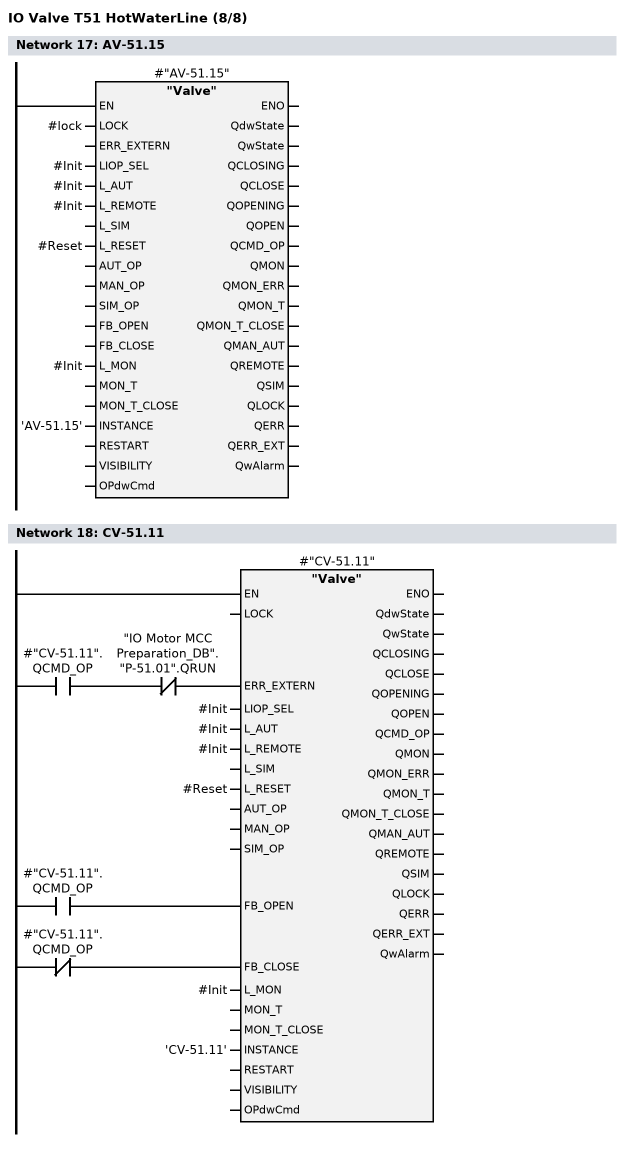
   RUNG wire#powerrail
      #"AV-51.15"(LOCK := #lock, ERR_EXTERN :=, LIOP_SEL := #Init, L_AUT := #Init, L_REMOTE := #Init, L_SIM :=, L_RESET := #Reset, AUT_OP :=, MAN_OP :=, SIM_OP :=, FB_OPEN :=, FB_CLOSE :=, L_MON := #Init, MON_T :=, MON_T_CLOSE :=, INSTANCE := 'AV-51.15', RESTART :=, VISIBILITY :=, OPdwCmd :=, QdwState =>, QwState =>, QCLOSING =>, QCLOSE =>, QOPENING =>, QOPEN =>, QCMD_OP =>, QMON =>, QMON_ERR =>, QMON_T =>, QMON_T_CLOSE =>, QMAN_AUT =>, QREMOTE =>, QSIM =>, QLOCK =>, QERR =>, QERR_EXT =>, QwAlarm =>)
   END_RUNG
   // the same network as SCL:
   #"AV-51.15"(LOCK := #lock,   // "Valve"
               LIOP_SEL := #Init,
               L_AUT := #Init,
               L_REMOTE := #Init,
               L_RESET := #Reset,
               L_MON := #Init,
               INSTANCE := 'AV-51.15');
END_REGION

REGION Network 18: CV-51.11
   RUNG wire#powerrail
      #"CV-51.11"(ERR_EXTERN := wire#w1, FB_OPEN := wire#w2, FB_CLOSE := wire#w3, LOCK :=, LIOP_SEL := #Init, L_AUT := #Init, L_REMOTE := #Init, L_SIM :=, L_RESET := #Reset, AUT_OP :=, MAN_OP :=, SIM_OP :=, L_MON := #Init, MON_T :=, MON_T_CLOSE :=, INSTANCE := 'CV-51.11', RESTART :=, VISIBILITY :=, OPdwCmd :=, QdwState =>, QwState =>, QCLOSING =>, QCLOSE =>, QOPENING =>, QOPEN =>, QCMD_OP =>, QMON =>, QMON_ERR =>, QMON_T =>, QMON_T_CLOSE =>, QMAN_AUT =>, QREMOTE =>, QSIM =>, QLOCK =>, QERR =>, QERR_EXT =>, QwAlarm =>)
   END_RUNG
   RUNG wire#powerrail
      Contact( #"CV-51.11".QCMD_OP )
      I_Contact( "IO Motor MCC Preparation_DB"."P-51.01".QRUN )
   END_RUNG wire#w1
   RUNG wire#powerrail
      Contact( #"CV-51.11".QCMD_OP )
   END_RUNG wire#w2
   RUNG wire#powerrail
      I_Contact( #"CV-51.11".QCMD_OP )
   END_RUNG wire#w3
   // the same network as SCL:
   #"CV-51.11"(ERR_EXTERN := #"CV-51.11".QCMD_OP AND NOT "IO Motor MCC Preparation_DB"."P-51.01".QRUN,   // "Valve"
               LIOP_SEL := #Init,
               L_AUT := #Init,
               L_REMOTE := #Init,
               L_RESET := #Reset,
               FB_OPEN := #"CV-51.11".QCMD_OP,
               FB_CLOSE := NOT #"CV-51.11".QCMD_OP,
               L_MON := #Init,
               INSTANCE := 'CV-51.11');
END_REGION
END_FUNCTION_BLOCK

FUNCTION "IO Homoge" : Void   // FC1, LAD
{ S7_Optimized_Access := 'TRUE' }
VERSION : 0.1
// stored: AutoNumber true, IsIECCheckEnabled false, SetENOAutomatically false, UDAEnableTagReadback false
BEGIN

REGION Network 1: Analog
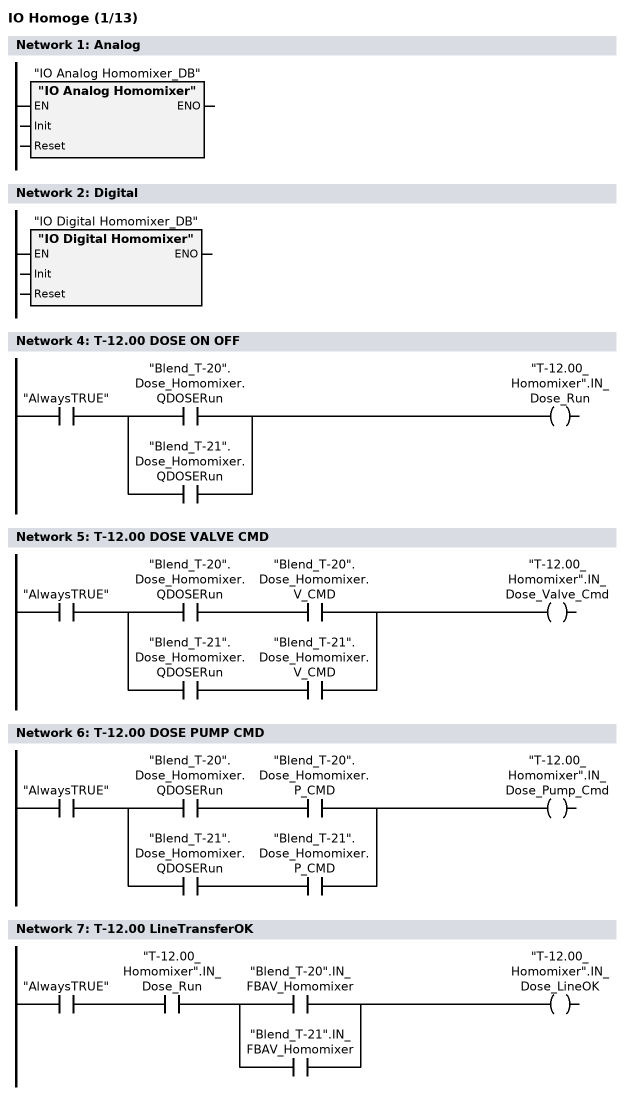
   RUNG wire#powerrail
      "IO Analog Homomixer_DB"(Init :=, Reset :=)
   END_RUNG
   // the same network as SCL:
   "IO Analog Homomixer_DB"();   // "IO Analog Homomixer"
END_REGION

REGION Network 2: Digital
   RUNG wire#powerrail
      "IO Digital Homomixer_DB"(Init :=, Reset :=)
   END_RUNG
   // the same network as SCL:
   "IO Digital Homomixer_DB"();   // "IO Digital Homomixer"
END_REGION

REGION Network 4: T-12.00 DOSE ON OFF
   RUNG wire#powerrail
      Contact( "AlwaysTRUE" )
      wire#w1
      Contact( "Blend_T-20".Dose_Homomixer.QDOSERun )
      wire#w2
      Coil( "T-12.00_Homomixer".IN_Dose_Run )
   END_RUNG
   RUNG wire#w1
      Contact( "Blend_T-21".Dose_Homomixer.QDOSERun )
   END_RUNG wire#w2
   // the same network as SCL:
   "T-12.00_Homomixer".IN_Dose_Run := "AlwaysTRUE" AND ("Blend_T-20".Dose_Homomixer.QDOSERun OR "Blend_T-21".Dose_Homomixer.QDOSERun);
END_REGION

REGION Network 5: T-12.00 DOSE VALVE CMD
   RUNG wire#powerrail
      Contact( "AlwaysTRUE" )
      wire#w1
      Contact( "Blend_T-20".Dose_Homomixer.QDOSERun )
      Contact( "Blend_T-20".Dose_Homomixer.V_CMD )
      wire#w2
      Coil( "T-12.00_Homomixer".IN_Dose_Valve_Cmd )
   END_RUNG
   RUNG wire#w1
      Contact( "Blend_T-21".Dose_Homomixer.QDOSERun )
      Contact( "Blend_T-21".Dose_Homomixer.V_CMD )
   END_RUNG wire#w2
   // the same network as SCL:
   "T-12.00_Homomixer".IN_Dose_Valve_Cmd := "AlwaysTRUE" AND (("Blend_T-20".Dose_Homomixer.QDOSERun AND "Blend_T-20".Dose_Homomixer.V_CMD) OR ("Blend_T-21".Dose_Homomixer.QDOSERun AND "Blend_T-21".Dose_Homomixer.V_CMD));
END_REGION

REGION Network 6: T-12.00 DOSE PUMP CMD
   RUNG wire#powerrail
      Contact( "AlwaysTRUE" )
      wire#w1
      Contact( "Blend_T-20".Dose_Homomixer.QDOSERun )
      Contact( "Blend_T-20".Dose_Homomixer.P_CMD )
      wire#w2
      Coil( "T-12.00_Homomixer".IN_Dose_Pump_Cmd )
   END_RUNG
   RUNG wire#w1
      Contact( "Blend_T-21".Dose_Homomixer.QDOSERun )
      Contact( "Blend_T-21".Dose_Homomixer.P_CMD )
   END_RUNG wire#w2
   // the same network as SCL:
   "T-12.00_Homomixer".IN_Dose_Pump_Cmd := "AlwaysTRUE" AND (("Blend_T-20".Dose_Homomixer.QDOSERun AND "Blend_T-20".Dose_Homomixer.P_CMD) OR ("Blend_T-21".Dose_Homomixer.QDOSERun AND "Blend_T-21".Dose_Homomixer.P_CMD));
END_REGION

REGION Network 7: T-12.00 LineTransferOK
   RUNG wire#powerrail
      Contact( "AlwaysTRUE" )
      Contact( "T-12.00_Homomixer".IN_Dose_Run )
      wire#w1
      Contact( "Blend_T-20".IN_FBAV_Homomixer )
      wire#w2
      Coil( "T-12.00_Homomixer".IN_Dose_LineOK )
   END_RUNG
   RUNG wire#w1
      Contact( "Blend_T-21".IN_FBAV_Homomixer )
   END_RUNG wire#w2
   // the same network as SCL:
   "T-12.00_Homomixer".IN_Dose_LineOK := "AlwaysTRUE" AND "T-12.00_Homomixer".IN_Dose_Run AND ("Blend_T-20".IN_FBAV_Homomixer OR "Blend_T-21".IN_FBAV_Homomixer);
END_REGION

REGION Network 8: T-12.00 Homomixer
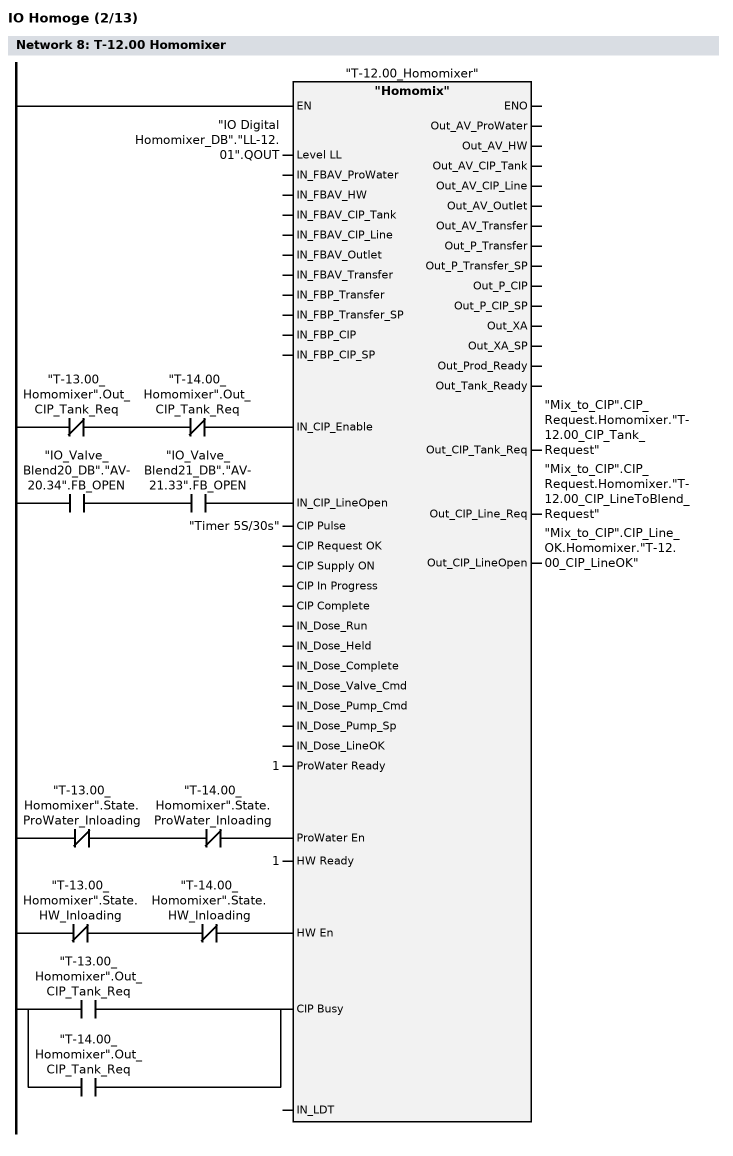
   RUNG wire#powerrail
      "T-12.00_Homomixer"(IN_CIP_Enable := wire#w1, IN_CIP_LineOpen := wire#w2, "ProWater En" := wire#w3, "HW En" := wire#w4, "CIP Busy" := wire#w5, "Level LL" := "IO Digital Homomixer_DB"."LL-12.01".QOUT, IN_FBAV_ProWater :=, IN_FBAV_HW :=, IN_FBAV_CIP_Tank :=, IN_FBAV_CIP_Line :=, IN_FBAV_Outlet :=, IN_FBAV_Transfer :=, IN_FBP_Transfer :=, IN_FBP_Transfer_SP :=, IN_FBP_CIP :=, IN_FBP_CIP_SP :=, "CIP Pulse" := "Timer 5S/30s", "CIP Request OK" :=, "CIP Supply ON" :=, "CIP In Progress" :=, "CIP Complete" :=, IN_Dose_Run :=, IN_Dose_Held :=, IN_Dose_Complete :=, IN_Dose_Valve_Cmd :=, IN_Dose_Pump_Cmd :=, IN_Dose_Pump_Sp :=, IN_Dose_LineOK :=, "ProWater Ready" := 1, "HW Ready" := 1, IN_LDT :=, Out_AV_ProWater =>, Out_AV_HW =>, Out_AV_CIP_Tank =>, Out_AV_CIP_Line =>, Out_AV_Outlet =>, Out_AV_Transfer =>, Out_P_Transfer =>, Out_P_Transfer_SP =>, Out_P_CIP =>, Out_P_CIP_SP =>, Out_XA =>, Out_XA_SP =>, Out_Prod_Ready =>, Out_Tank_Ready =>, Out_CIP_Tank_Req => "Mix_to_CIP".CIP_Request.Homomixer."T-12.00_CIP_Tank_Request", Out_CIP_Line_Req => "Mix_to_CIP".CIP_Request.Homomixer."T-12.00_CIP_LineToBlend_Request", Out_CIP_LineOpen => "Mix_to_CIP".CIP_Line_OK.Homomixer."T-12.00_CIP_LineOK")
   END_RUNG
   RUNG wire#powerrail
      I_Contact( "T-13.00_Homomixer".Out_CIP_Tank_Req )
      I_Contact( "T-14.00_Homomixer".Out_CIP_Tank_Req )
   END_RUNG wire#w1
   RUNG wire#powerrail
      Contact( "IO_Valve_Blend20_DB"."AV-20.34".FB_OPEN )
      Contact( "IO_Valve_Blend21_DB"."AV-21.33".FB_OPEN )
   END_RUNG wire#w2
   RUNG wire#powerrail
      I_Contact( "T-13.00_Homomixer".State.ProWater_Inloading )
      I_Contact( "T-14.00_Homomixer".State.ProWater_Inloading )
   END_RUNG wire#w3
   RUNG wire#powerrail
      I_Contact( "T-13.00_Homomixer".State.HW_Inloading )
      I_Contact( "T-14.00_Homomixer".State.HW_Inloading )
   END_RUNG wire#w4
   RUNG wire#powerrail
      Contact( "T-13.00_Homomixer".Out_CIP_Tank_Req )
   END_RUNG wire#w5
   RUNG wire#powerrail
      Contact( "T-14.00_Homomixer".Out_CIP_Tank_Req )
   END_RUNG wire#w5
   // the same network as SCL:
   "T-12.00_Homomixer"("Level LL" := "IO Digital Homomixer_DB"."LL-12.01".QOUT,   // "Homomix"
                       IN_CIP_Enable := NOT "T-13.00_Homomixer".Out_CIP_Tank_Req AND NOT "T-14.00_Homomixer".Out_CIP_Tank_Req,
                       IN_CIP_LineOpen := "IO_Valve_Blend20_DB"."AV-20.34".FB_OPEN AND "IO_Valve_Blend21_DB"."AV-21.33".FB_OPEN,
                       "CIP Pulse" := "Timer 5S/30s",
                       "ProWater Ready" := 1,
                       "ProWater En" := NOT "T-13.00_Homomixer".State.ProWater_Inloading AND NOT "T-14.00_Homomixer".State.ProWater_Inloading,
                       "HW Ready" := 1,
                       "HW En" := NOT "T-13.00_Homomixer".State.HW_Inloading AND NOT "T-14.00_Homomixer".State.HW_Inloading,
                       "CIP Busy" := "T-13.00_Homomixer".Out_CIP_Tank_Req OR "T-14.00_Homomixer".Out_CIP_Tank_Req,
                       Out_CIP_Tank_Req => "Mix_to_CIP".CIP_Request.Homomixer."T-12.00_CIP_Tank_Request",
                       Out_CIP_Line_Req => "Mix_to_CIP".CIP_Request.Homomixer."T-12.00_CIP_LineToBlend_Request",
                       Out_CIP_LineOpen => "Mix_to_CIP".CIP_Line_OK.Homomixer."T-12.00_CIP_LineOK");
END_REGION

REGION Network 9: T-12.00 Valve Cmd
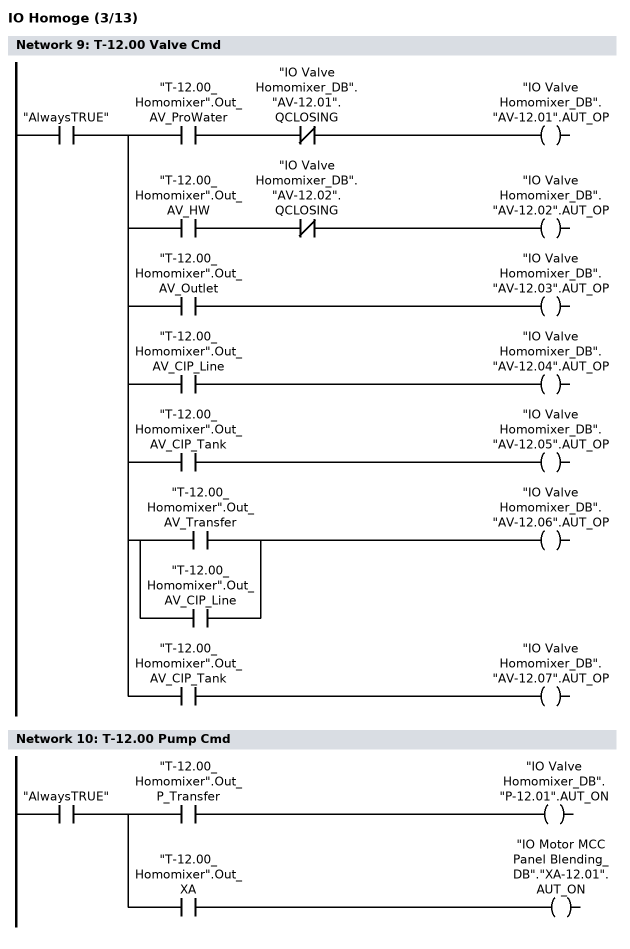
   RUNG wire#powerrail
      Contact( "AlwaysTRUE" )
      wire#w1
      Contact( "T-12.00_Homomixer".Out_AV_ProWater )
      I_Contact( "IO Valve Homomixer_DB"."AV-12.01".QCLOSING )
      Coil( "IO Valve Homomixer_DB"."AV-12.01".AUT_OP )
   END_RUNG
   RUNG wire#w1
      Contact( "T-12.00_Homomixer".Out_AV_HW )
      I_Contact( "IO Valve Homomixer_DB"."AV-12.02".QCLOSING )
      Coil( "IO Valve Homomixer_DB"."AV-12.02".AUT_OP )
   END_RUNG
   RUNG wire#w1
      Contact( "T-12.00_Homomixer".Out_AV_Outlet )
      Coil( "IO Valve Homomixer_DB"."AV-12.03".AUT_OP )
   END_RUNG
   RUNG wire#w1
      Contact( "T-12.00_Homomixer".Out_AV_CIP_Line )
      Coil( "IO Valve Homomixer_DB"."AV-12.04".AUT_OP )
   END_RUNG
   RUNG wire#w1
      Contact( "T-12.00_Homomixer".Out_AV_CIP_Tank )
      Coil( "IO Valve Homomixer_DB"."AV-12.05".AUT_OP )
   END_RUNG
   RUNG wire#w1
      Contact( "T-12.00_Homomixer".Out_AV_Transfer )
      wire#w2
      Coil( "IO Valve Homomixer_DB"."AV-12.06".AUT_OP )
   END_RUNG
   RUNG wire#w1
      Contact( "T-12.00_Homomixer".Out_AV_CIP_Line )
   END_RUNG wire#w2
   RUNG wire#w1
      Contact( "T-12.00_Homomixer".Out_AV_CIP_Tank )
      Coil( "IO Valve Homomixer_DB"."AV-12.07".AUT_OP )
   END_RUNG
   // the same network as SCL:
   "IO Valve Homomixer_DB"."AV-12.01".AUT_OP := "AlwaysTRUE" AND "T-12.00_Homomixer".Out_AV_ProWater AND NOT "IO Valve Homomixer_DB"."AV-12.01".QCLOSING;
   "IO Valve Homomixer_DB"."AV-12.02".AUT_OP := "AlwaysTRUE" AND "T-12.00_Homomixer".Out_AV_HW AND NOT "IO Valve Homomixer_DB"."AV-12.02".QCLOSING;
   "IO Valve Homomixer_DB"."AV-12.03".AUT_OP := "AlwaysTRUE" AND "T-12.00_Homomixer".Out_AV_Outlet;
   "IO Valve Homomixer_DB"."AV-12.04".AUT_OP := "AlwaysTRUE" AND "T-12.00_Homomixer".Out_AV_CIP_Line;
   "IO Valve Homomixer_DB"."AV-12.05".AUT_OP := "AlwaysTRUE" AND "T-12.00_Homomixer".Out_AV_CIP_Tank;
   "IO Valve Homomixer_DB"."AV-12.06".AUT_OP := "AlwaysTRUE" AND ("T-12.00_Homomixer".Out_AV_Transfer OR "T-12.00_Homomixer".Out_AV_CIP_Line);
   "IO Valve Homomixer_DB"."AV-12.07".AUT_OP := "AlwaysTRUE" AND "T-12.00_Homomixer".Out_AV_CIP_Tank;
END_REGION

REGION Network 10: T-12.00 Pump Cmd
   RUNG wire#powerrail
      Contact( "AlwaysTRUE" )
      wire#w1
      Contact( "T-12.00_Homomixer".Out_P_Transfer )
      Coil( "IO Valve Homomixer_DB"."P-12.01".AUT_ON )
   END_RUNG
   RUNG wire#w1
      Contact( "T-12.00_Homomixer".Out_XA )
      Coil( "IO Motor MCC Panel Blending_DB"."XA-12.01".AUT_ON )
   END_RUNG
   // the same network as SCL:
   "IO Valve Homomixer_DB"."P-12.01".AUT_ON := "AlwaysTRUE" AND "T-12.00_Homomixer".Out_P_Transfer;
   "IO Motor MCC Panel Blending_DB"."XA-12.01".AUT_ON := "AlwaysTRUE" AND "T-12.00_Homomixer".Out_XA;
END_REGION

REGION Network 11: T-12.00 Feedback Instrument
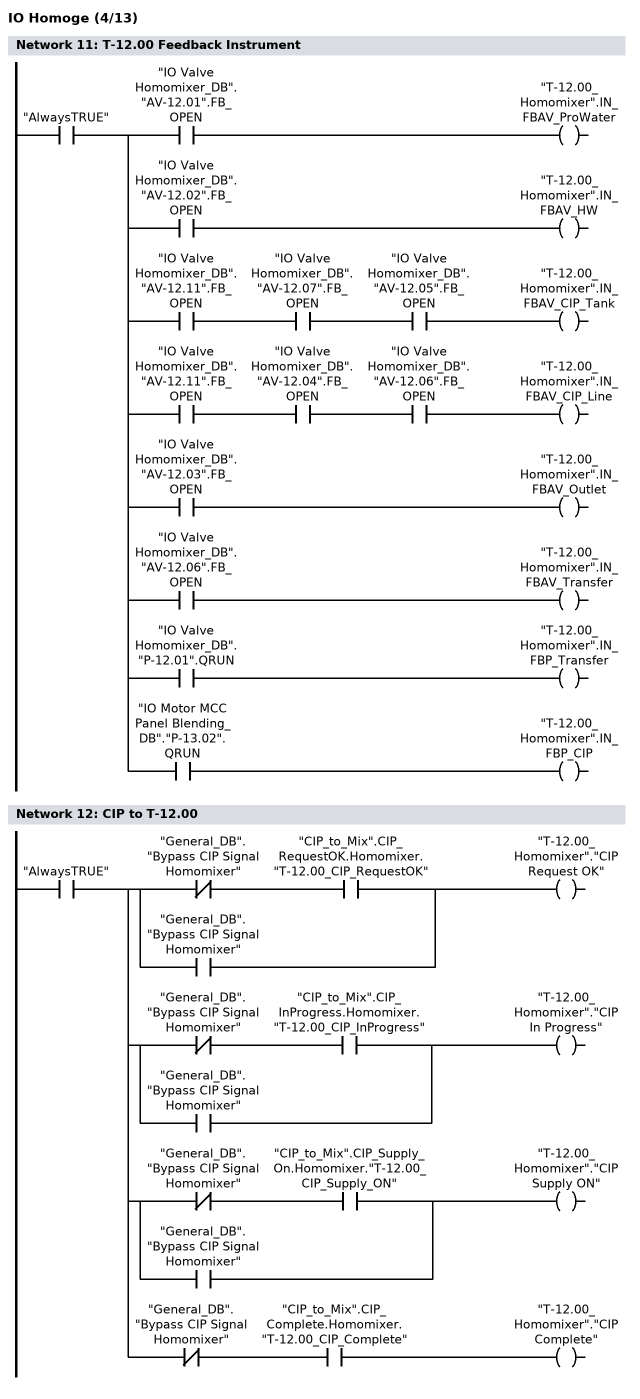
   RUNG wire#powerrail
      Contact( "AlwaysTRUE" )
      wire#w1
      Contact( "IO Valve Homomixer_DB"."AV-12.01".FB_OPEN )
      Coil( "T-12.00_Homomixer".IN_FBAV_ProWater )
   END_RUNG
   RUNG wire#w1
      Contact( "IO Valve Homomixer_DB"."AV-12.02".FB_OPEN )
      Coil( "T-12.00_Homomixer".IN_FBAV_HW )
   END_RUNG
   RUNG wire#w1
      Contact( "IO Valve Homomixer_DB"."AV-12.11".FB_OPEN )
      Contact( "IO Valve Homomixer_DB"."AV-12.07".FB_OPEN )
      Contact( "IO Valve Homomixer_DB"."AV-12.05".FB_OPEN )
      Coil( "T-12.00_Homomixer".IN_FBAV_CIP_Tank )
   END_RUNG
   RUNG wire#w1
      Contact( "IO Valve Homomixer_DB"."AV-12.11".FB_OPEN )
      Contact( "IO Valve Homomixer_DB"."AV-12.04".FB_OPEN )
      Contact( "IO Valve Homomixer_DB"."AV-12.06".FB_OPEN )
      Coil( "T-12.00_Homomixer".IN_FBAV_CIP_Line )
   END_RUNG
   RUNG wire#w1
      Contact( "IO Valve Homomixer_DB"."AV-12.03".FB_OPEN )
      Coil( "T-12.00_Homomixer".IN_FBAV_Outlet )
   END_RUNG
   RUNG wire#w1
      Contact( "IO Valve Homomixer_DB"."AV-12.06".FB_OPEN )
      Coil( "T-12.00_Homomixer".IN_FBAV_Transfer )
   END_RUNG
   RUNG wire#w1
      Contact( "IO Valve Homomixer_DB"."P-12.01".QRUN )
      Coil( "T-12.00_Homomixer".IN_FBP_Transfer )
   END_RUNG
   RUNG wire#w1
      Contact( "IO Motor MCC Panel Blending_DB"."P-13.02".QRUN )
      Coil( "T-12.00_Homomixer".IN_FBP_CIP )
   END_RUNG
   // the same network as SCL:
   "T-12.00_Homomixer".IN_FBAV_ProWater := "AlwaysTRUE" AND "IO Valve Homomixer_DB"."AV-12.01".FB_OPEN;
   "T-12.00_Homomixer".IN_FBAV_HW := "AlwaysTRUE" AND "IO Valve Homomixer_DB"."AV-12.02".FB_OPEN;
   "T-12.00_Homomixer".IN_FBAV_CIP_Tank := "AlwaysTRUE" AND "IO Valve Homomixer_DB"."AV-12.11".FB_OPEN AND "IO Valve Homomixer_DB"."AV-12.07".FB_OPEN AND "IO Valve Homomixer_DB"."AV-12.05".FB_OPEN;
   "T-12.00_Homomixer".IN_FBAV_CIP_Line := "AlwaysTRUE" AND "IO Valve Homomixer_DB"."AV-12.11".FB_OPEN AND "IO Valve Homomixer_DB"."AV-12.04".FB_OPEN AND "IO Valve Homomixer_DB"."AV-12.06".FB_OPEN;
   "T-12.00_Homomixer".IN_FBAV_Outlet := "AlwaysTRUE" AND "IO Valve Homomixer_DB"."AV-12.03".FB_OPEN;
   "T-12.00_Homomixer".IN_FBAV_Transfer := "AlwaysTRUE" AND "IO Valve Homomixer_DB"."AV-12.06".FB_OPEN;
   "T-12.00_Homomixer".IN_FBP_Transfer := "AlwaysTRUE" AND "IO Valve Homomixer_DB"."P-12.01".QRUN;
   "T-12.00_Homomixer".IN_FBP_CIP := "AlwaysTRUE" AND "IO Motor MCC Panel Blending_DB"."P-13.02".QRUN;
END_REGION

REGION Network 12: CIP to T-12.00
   RUNG wire#powerrail
      Contact( "AlwaysTRUE" )
      wire#w1
      I_Contact( "General_DB"."Bypass CIP Signal Homomixer" )
      Contact( "CIP_to_Mix".CIP_RequestOK.Homomixer."T-12.00_CIP_RequestOK" )
      wire#w2
      Coil( "T-12.00_Homomixer"."CIP Request OK" )
   END_RUNG
   RUNG wire#w1
      Contact( "General_DB"."Bypass CIP Signal Homomixer" )
   END_RUNG wire#w2
   RUNG wire#w1
      I_Contact( "General_DB"."Bypass CIP Signal Homomixer" )
      Contact( "CIP_to_Mix".CIP_InProgress.Homomixer."T-12.00_CIP_InProgress" )
      wire#w3
      Coil( "T-12.00_Homomixer"."CIP In Progress" )
   END_RUNG
   RUNG wire#w1
      Contact( "General_DB"."Bypass CIP Signal Homomixer" )
   END_RUNG wire#w3
   RUNG wire#w1
      I_Contact( "General_DB"."Bypass CIP Signal Homomixer" )
      Contact( "CIP_to_Mix".CIP_Supply_On.Homomixer."T-12.00_CIP_Supply_ON" )
      wire#w4
      Coil( "T-12.00_Homomixer"."CIP Supply ON" )
   END_RUNG
   RUNG wire#w1
      Contact( "General_DB"."Bypass CIP Signal Homomixer" )
   END_RUNG wire#w4
   RUNG wire#w1
      I_Contact( "General_DB"."Bypass CIP Signal Homomixer" )
      Contact( "CIP_to_Mix".CIP_Complete.Homomixer."T-12.00_CIP_Complete" )
      Coil( "T-12.00_Homomixer"."CIP Complete" )
   END_RUNG
   // the same network as SCL:
   "T-12.00_Homomixer"."CIP Request OK" := "AlwaysTRUE" AND ((NOT "General_DB"."Bypass CIP Signal Homomixer" AND "CIP_to_Mix".CIP_RequestOK.Homomixer."T-12.00_CIP_RequestOK") OR "General_DB"."Bypass CIP Signal Homomixer");
   "T-12.00_Homomixer"."CIP In Progress" := "AlwaysTRUE" AND ((NOT "General_DB"."Bypass CIP Signal Homomixer" AND "CIP_to_Mix".CIP_InProgress.Homomixer."T-12.00_CIP_InProgress") OR "General_DB"."Bypass CIP Signal Homomixer");
   "T-12.00_Homomixer"."CIP Supply ON" := "AlwaysTRUE" AND ((NOT "General_DB"."Bypass CIP Signal Homomixer" AND "CIP_to_Mix".CIP_Supply_On.Homomixer."T-12.00_CIP_Supply_ON") OR "General_DB"."Bypass CIP Signal Homomixer");
   "T-12.00_Homomixer"."CIP Complete" := "AlwaysTRUE" AND NOT "General_DB"."Bypass CIP Signal Homomixer" AND "CIP_to_Mix".CIP_Complete.Homomixer."T-12.00_CIP_Complete";
END_REGION

REGION Network 15: T-13.00 DOSE ON OFF
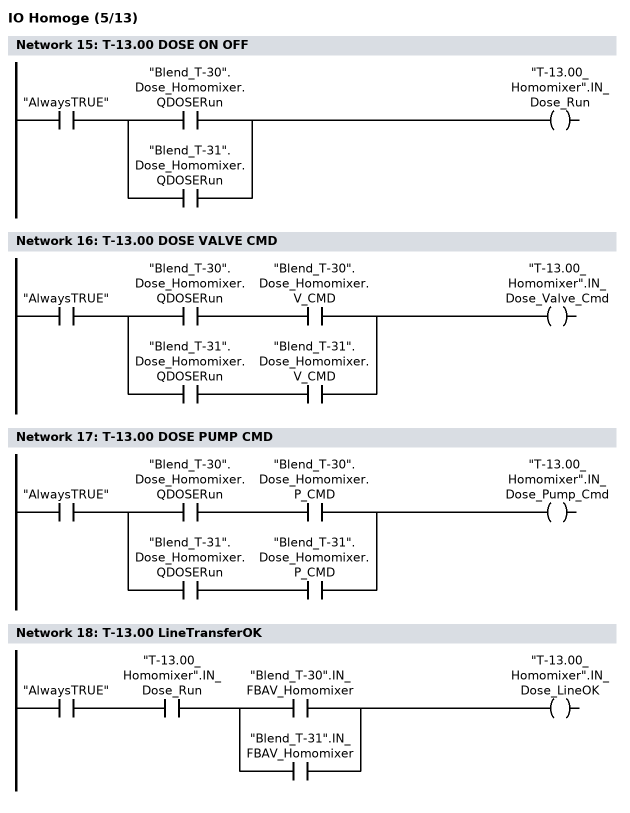
   RUNG wire#powerrail
      Contact( "AlwaysTRUE" )
      wire#w1
      Contact( "Blend_T-30".Dose_Homomixer.QDOSERun )
      wire#w2
      Coil( "T-13.00_Homomixer".IN_Dose_Run )
   END_RUNG
   RUNG wire#w1
      Contact( "Blend_T-31".Dose_Homomixer.QDOSERun )
   END_RUNG wire#w2
   // the same network as SCL:
   "T-13.00_Homomixer".IN_Dose_Run := "AlwaysTRUE" AND ("Blend_T-30".Dose_Homomixer.QDOSERun OR "Blend_T-31".Dose_Homomixer.QDOSERun);
END_REGION

REGION Network 16: T-13.00 DOSE VALVE CMD
   RUNG wire#powerrail
      Contact( "AlwaysTRUE" )
      wire#w1
      Contact( "Blend_T-30".Dose_Homomixer.QDOSERun )
      Contact( "Blend_T-30".Dose_Homomixer.V_CMD )
      wire#w2
      Coil( "T-13.00_Homomixer".IN_Dose_Valve_Cmd )
   END_RUNG
   RUNG wire#w1
      Contact( "Blend_T-31".Dose_Homomixer.QDOSERun )
      Contact( "Blend_T-31".Dose_Homomixer.V_CMD )
   END_RUNG wire#w2
   // the same network as SCL:
   "T-13.00_Homomixer".IN_Dose_Valve_Cmd := "AlwaysTRUE" AND (("Blend_T-30".Dose_Homomixer.QDOSERun AND "Blend_T-30".Dose_Homomixer.V_CMD) OR ("Blend_T-31".Dose_Homomixer.QDOSERun AND "Blend_T-31".Dose_Homomixer.V_CMD));
END_REGION

REGION Network 17: T-13.00 DOSE PUMP CMD
   RUNG wire#powerrail
      Contact( "AlwaysTRUE" )
      wire#w1
      Contact( "Blend_T-30".Dose_Homomixer.QDOSERun )
      Contact( "Blend_T-30".Dose_Homomixer.P_CMD )
      wire#w2
      Coil( "T-13.00_Homomixer".IN_Dose_Pump_Cmd )
   END_RUNG
   RUNG wire#w1
      Contact( "Blend_T-31".Dose_Homomixer.QDOSERun )
      Contact( "Blend_T-31".Dose_Homomixer.P_CMD )
   END_RUNG wire#w2
   // the same network as SCL:
   "T-13.00_Homomixer".IN_Dose_Pump_Cmd := "AlwaysTRUE" AND (("Blend_T-30".Dose_Homomixer.QDOSERun AND "Blend_T-30".Dose_Homomixer.P_CMD) OR ("Blend_T-31".Dose_Homomixer.QDOSERun AND "Blend_T-31".Dose_Homomixer.P_CMD));
END_REGION

REGION Network 18: T-13.00 LineTransferOK
   RUNG wire#powerrail
      Contact( "AlwaysTRUE" )
      Contact( "T-13.00_Homomixer".IN_Dose_Run )
      wire#w1
      Contact( "Blend_T-30".IN_FBAV_Homomixer )
      wire#w2
      Coil( "T-13.00_Homomixer".IN_Dose_LineOK )
   END_RUNG
   RUNG wire#w1
      Contact( "Blend_T-31".IN_FBAV_Homomixer )
   END_RUNG wire#w2
   // the same network as SCL:
   "T-13.00_Homomixer".IN_Dose_LineOK := "AlwaysTRUE" AND "T-13.00_Homomixer".IN_Dose_Run AND ("Blend_T-30".IN_FBAV_Homomixer OR "Blend_T-31".IN_FBAV_Homomixer);
END_REGION

REGION Network 19: T-13.00 Homomixer
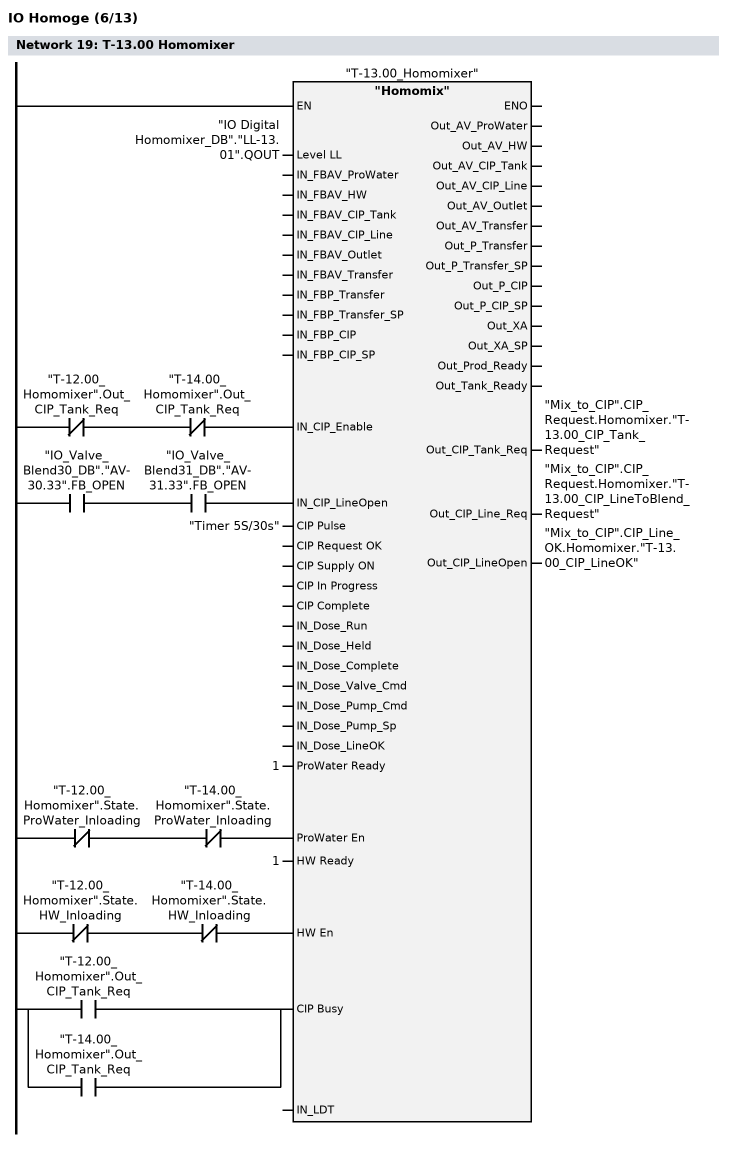
   RUNG wire#powerrail
      "T-13.00_Homomixer"(IN_CIP_Enable := wire#w1, IN_CIP_LineOpen := wire#w2, "ProWater En" := wire#w3, "HW En" := wire#w4, "CIP Busy" := wire#w5, "Level LL" := "IO Digital Homomixer_DB"."LL-13.01".QOUT, IN_FBAV_ProWater :=, IN_FBAV_HW :=, IN_FBAV_CIP_Tank :=, IN_FBAV_CIP_Line :=, IN_FBAV_Outlet :=, IN_FBAV_Transfer :=, IN_FBP_Transfer :=, IN_FBP_Transfer_SP :=, IN_FBP_CIP :=, IN_FBP_CIP_SP :=, "CIP Pulse" := "Timer 5S/30s", "CIP Request OK" :=, "CIP Supply ON" :=, "CIP In Progress" :=, "CIP Complete" :=, IN_Dose_Run :=, IN_Dose_Held :=, IN_Dose_Complete :=, IN_Dose_Valve_Cmd :=, IN_Dose_Pump_Cmd :=, IN_Dose_Pump_Sp :=, IN_Dose_LineOK :=, "ProWater Ready" := 1, "HW Ready" := 1, IN_LDT :=, Out_AV_ProWater =>, Out_AV_HW =>, Out_AV_CIP_Tank =>, Out_AV_CIP_Line =>, Out_AV_Outlet =>, Out_AV_Transfer =>, Out_P_Transfer =>, Out_P_Transfer_SP =>, Out_P_CIP =>, Out_P_CIP_SP =>, Out_XA =>, Out_XA_SP =>, Out_Prod_Ready =>, Out_Tank_Ready =>, Out_CIP_Tank_Req => "Mix_to_CIP".CIP_Request.Homomixer."T-13.00_CIP_Tank_Request", Out_CIP_Line_Req => "Mix_to_CIP".CIP_Request.Homomixer."T-13.00_CIP_LineToBlend_Request", Out_CIP_LineOpen => "Mix_to_CIP".CIP_Line_OK.Homomixer."T-13.00_CIP_LineOK")
   END_RUNG
   RUNG wire#powerrail
      I_Contact( "T-12.00_Homomixer".Out_CIP_Tank_Req )
      I_Contact( "T-14.00_Homomixer".Out_CIP_Tank_Req )
   END_RUNG wire#w1
   RUNG wire#powerrail
      Contact( "IO_Valve_Blend30_DB"."AV-30.33".FB_OPEN )
      Contact( "IO_Valve_Blend31_DB"."AV-31.33".FB_OPEN )
   END_RUNG wire#w2
   RUNG wire#powerrail
      I_Contact( "T-12.00_Homomixer".State.ProWater_Inloading )
      I_Contact( "T-14.00_Homomixer".State.ProWater_Inloading )
   END_RUNG wire#w3
   RUNG wire#powerrail
      I_Contact( "T-12.00_Homomixer".State.HW_Inloading )
      I_Contact( "T-14.00_Homomixer".State.HW_Inloading )
   END_RUNG wire#w4
   RUNG wire#powerrail
      Contact( "T-12.00_Homomixer".Out_CIP_Tank_Req )
   END_RUNG wire#w5
   RUNG wire#powerrail
      Contact( "T-14.00_Homomixer".Out_CIP_Tank_Req )
   END_RUNG wire#w5
   // the same network as SCL:
   "T-13.00_Homomixer"("Level LL" := "IO Digital Homomixer_DB"."LL-13.01".QOUT,   // "Homomix"
                       IN_CIP_Enable := NOT "T-12.00_Homomixer".Out_CIP_Tank_Req AND NOT "T-14.00_Homomixer".Out_CIP_Tank_Req,
                       IN_CIP_LineOpen := "IO_Valve_Blend30_DB"."AV-30.33".FB_OPEN AND "IO_Valve_Blend31_DB"."AV-31.33".FB_OPEN,
                       "CIP Pulse" := "Timer 5S/30s",
                       "ProWater Ready" := 1,
                       "ProWater En" := NOT "T-12.00_Homomixer".State.ProWater_Inloading AND NOT "T-14.00_Homomixer".State.ProWater_Inloading,
                       "HW Ready" := 1,
                       "HW En" := NOT "T-12.00_Homomixer".State.HW_Inloading AND NOT "T-14.00_Homomixer".State.HW_Inloading,
                       "CIP Busy" := "T-12.00_Homomixer".Out_CIP_Tank_Req OR "T-14.00_Homomixer".Out_CIP_Tank_Req,
                       Out_CIP_Tank_Req => "Mix_to_CIP".CIP_Request.Homomixer."T-13.00_CIP_Tank_Request",
                       Out_CIP_Line_Req => "Mix_to_CIP".CIP_Request.Homomixer."T-13.00_CIP_LineToBlend_Request",
                       Out_CIP_LineOpen => "Mix_to_CIP".CIP_Line_OK.Homomixer."T-13.00_CIP_LineOK");
END_REGION

REGION Network 20: T-13.00 Valve Cmd
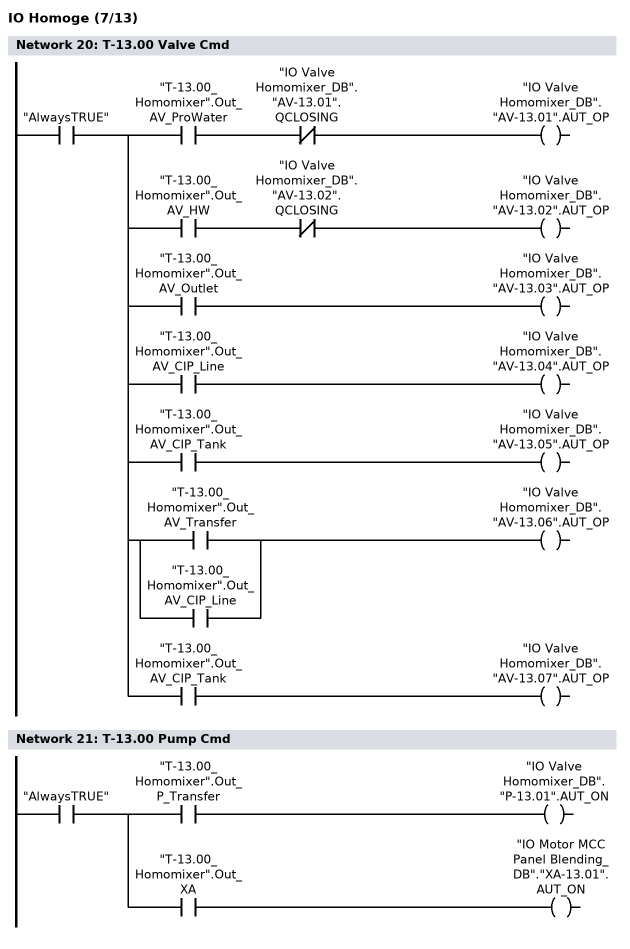
   RUNG wire#powerrail
      Contact( "AlwaysTRUE" )
      wire#w1
      Contact( "T-13.00_Homomixer".Out_AV_ProWater )
      I_Contact( "IO Valve Homomixer_DB"."AV-13.01".QCLOSING )
      Coil( "IO Valve Homomixer_DB"."AV-13.01".AUT_OP )
   END_RUNG
   RUNG wire#w1
      Contact( "T-13.00_Homomixer".Out_AV_HW )
      I_Contact( "IO Valve Homomixer_DB"."AV-13.02".QCLOSING )
      Coil( "IO Valve Homomixer_DB"."AV-13.02".AUT_OP )
   END_RUNG
   RUNG wire#w1
      Contact( "T-13.00_Homomixer".Out_AV_Outlet )
      Coil( "IO Valve Homomixer_DB"."AV-13.03".AUT_OP )
   END_RUNG
   RUNG wire#w1
      Contact( "T-13.00_Homomixer".Out_AV_CIP_Line )
      Coil( "IO Valve Homomixer_DB"."AV-13.04".AUT_OP )
   END_RUNG
   RUNG wire#w1
      Contact( "T-13.00_Homomixer".Out_AV_CIP_Tank )
      Coil( "IO Valve Homomixer_DB"."AV-13.05".AUT_OP )
   END_RUNG
   RUNG wire#w1
      Contact( "T-13.00_Homomixer".Out_AV_Transfer )
      wire#w2
      Coil( "IO Valve Homomixer_DB"."AV-13.06".AUT_OP )
   END_RUNG
   RUNG wire#w1
      Contact( "T-13.00_Homomixer".Out_AV_CIP_Line )
   END_RUNG wire#w2
   RUNG wire#w1
      Contact( "T-13.00_Homomixer".Out_AV_CIP_Tank )
      Coil( "IO Valve Homomixer_DB"."AV-13.07".AUT_OP )
   END_RUNG
   // the same network as SCL:
   "IO Valve Homomixer_DB"."AV-13.01".AUT_OP := "AlwaysTRUE" AND "T-13.00_Homomixer".Out_AV_ProWater AND NOT "IO Valve Homomixer_DB"."AV-13.01".QCLOSING;
   "IO Valve Homomixer_DB"."AV-13.02".AUT_OP := "AlwaysTRUE" AND "T-13.00_Homomixer".Out_AV_HW AND NOT "IO Valve Homomixer_DB"."AV-13.02".QCLOSING;
   "IO Valve Homomixer_DB"."AV-13.03".AUT_OP := "AlwaysTRUE" AND "T-13.00_Homomixer".Out_AV_Outlet;
   "IO Valve Homomixer_DB"."AV-13.04".AUT_OP := "AlwaysTRUE" AND "T-13.00_Homomixer".Out_AV_CIP_Line;
   "IO Valve Homomixer_DB"."AV-13.05".AUT_OP := "AlwaysTRUE" AND "T-13.00_Homomixer".Out_AV_CIP_Tank;
   "IO Valve Homomixer_DB"."AV-13.06".AUT_OP := "AlwaysTRUE" AND ("T-13.00_Homomixer".Out_AV_Transfer OR "T-13.00_Homomixer".Out_AV_CIP_Line);
   "IO Valve Homomixer_DB"."AV-13.07".AUT_OP := "AlwaysTRUE" AND "T-13.00_Homomixer".Out_AV_CIP_Tank;
END_REGION

REGION Network 21: T-13.00 Pump Cmd
   RUNG wire#powerrail
      Contact( "AlwaysTRUE" )
      wire#w1
      Contact( "T-13.00_Homomixer".Out_P_Transfer )
      Coil( "IO Valve Homomixer_DB"."P-13.01".AUT_ON )
   END_RUNG
   RUNG wire#w1
      Contact( "T-13.00_Homomixer".Out_XA )
      Coil( "IO Motor MCC Panel Blending_DB"."XA-13.01".AUT_ON )
   END_RUNG
   // the same network as SCL:
   "IO Valve Homomixer_DB"."P-13.01".AUT_ON := "AlwaysTRUE" AND "T-13.00_Homomixer".Out_P_Transfer;
   "IO Motor MCC Panel Blending_DB"."XA-13.01".AUT_ON := "AlwaysTRUE" AND "T-13.00_Homomixer".Out_XA;
END_REGION

REGION Network 22: T-13.00 Feedback Instrument
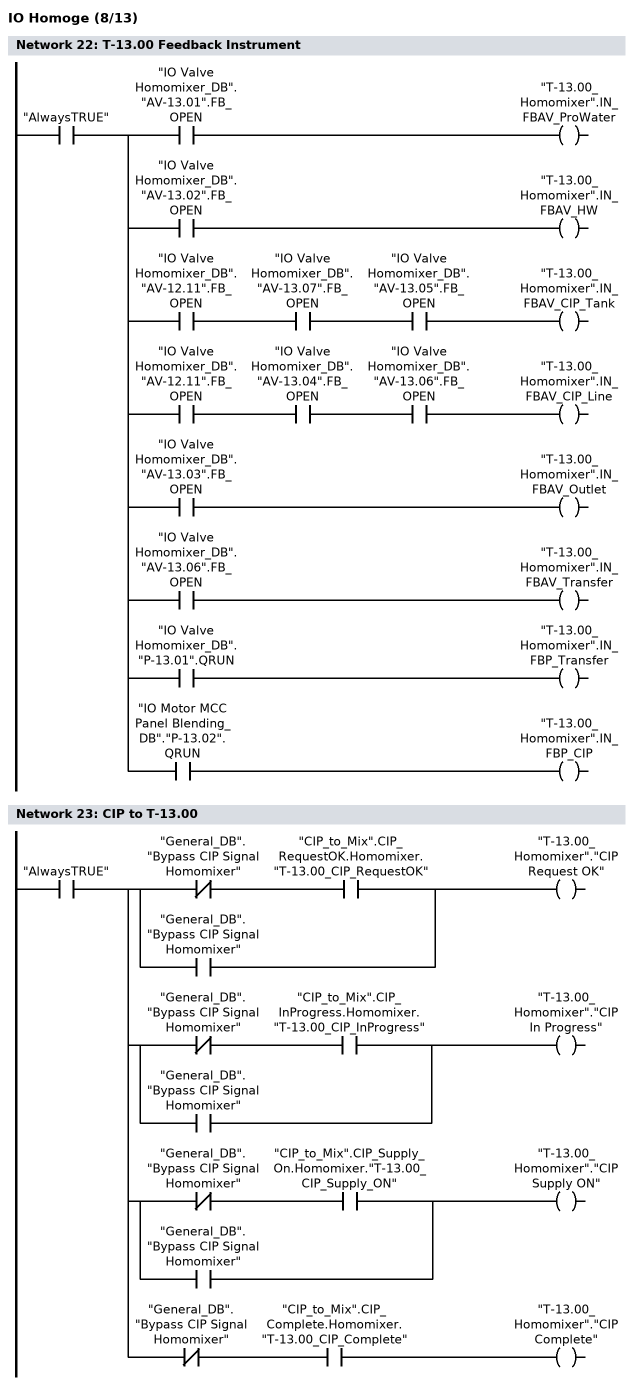
   RUNG wire#powerrail
      Contact( "AlwaysTRUE" )
      wire#w1
      Contact( "IO Valve Homomixer_DB"."AV-13.01".FB_OPEN )
      Coil( "T-13.00_Homomixer".IN_FBAV_ProWater )
   END_RUNG
   RUNG wire#w1
      Contact( "IO Valve Homomixer_DB"."AV-13.02".FB_OPEN )
      Coil( "T-13.00_Homomixer".IN_FBAV_HW )
   END_RUNG
   RUNG wire#w1
      Contact( "IO Valve Homomixer_DB"."AV-12.11".FB_OPEN )
      Contact( "IO Valve Homomixer_DB"."AV-13.07".FB_OPEN )
      Contact( "IO Valve Homomixer_DB"."AV-13.05".FB_OPEN )
      Coil( "T-13.00_Homomixer".IN_FBAV_CIP_Tank )
   END_RUNG
   RUNG wire#w1
      Contact( "IO Valve Homomixer_DB"."AV-12.11".FB_OPEN )
      Contact( "IO Valve Homomixer_DB"."AV-13.04".FB_OPEN )
      Contact( "IO Valve Homomixer_DB"."AV-13.06".FB_OPEN )
      Coil( "T-13.00_Homomixer".IN_FBAV_CIP_Line )
   END_RUNG
   RUNG wire#w1
      Contact( "IO Valve Homomixer_DB"."AV-13.03".FB_OPEN )
      Coil( "T-13.00_Homomixer".IN_FBAV_Outlet )
   END_RUNG
   RUNG wire#w1
      Contact( "IO Valve Homomixer_DB"."AV-13.06".FB_OPEN )
      Coil( "T-13.00_Homomixer".IN_FBAV_Transfer )
   END_RUNG
   RUNG wire#w1
      Contact( "IO Valve Homomixer_DB"."P-13.01".QRUN )
      Coil( "T-13.00_Homomixer".IN_FBP_Transfer )
   END_RUNG
   RUNG wire#w1
      Contact( "IO Motor MCC Panel Blending_DB"."P-13.02".QRUN )
      Coil( "T-13.00_Homomixer".IN_FBP_CIP )
   END_RUNG
   // the same network as SCL:
   "T-13.00_Homomixer".IN_FBAV_ProWater := "AlwaysTRUE" AND "IO Valve Homomixer_DB"."AV-13.01".FB_OPEN;
   "T-13.00_Homomixer".IN_FBAV_HW := "AlwaysTRUE" AND "IO Valve Homomixer_DB"."AV-13.02".FB_OPEN;
   "T-13.00_Homomixer".IN_FBAV_CIP_Tank := "AlwaysTRUE" AND "IO Valve Homomixer_DB"."AV-12.11".FB_OPEN AND "IO Valve Homomixer_DB"."AV-13.07".FB_OPEN AND "IO Valve Homomixer_DB"."AV-13.05".FB_OPEN;
   "T-13.00_Homomixer".IN_FBAV_CIP_Line := "AlwaysTRUE" AND "IO Valve Homomixer_DB"."AV-12.11".FB_OPEN AND "IO Valve Homomixer_DB"."AV-13.04".FB_OPEN AND "IO Valve Homomixer_DB"."AV-13.06".FB_OPEN;
   "T-13.00_Homomixer".IN_FBAV_Outlet := "AlwaysTRUE" AND "IO Valve Homomixer_DB"."AV-13.03".FB_OPEN;
   "T-13.00_Homomixer".IN_FBAV_Transfer := "AlwaysTRUE" AND "IO Valve Homomixer_DB"."AV-13.06".FB_OPEN;
   "T-13.00_Homomixer".IN_FBP_Transfer := "AlwaysTRUE" AND "IO Valve Homomixer_DB"."P-13.01".QRUN;
   "T-13.00_Homomixer".IN_FBP_CIP := "AlwaysTRUE" AND "IO Motor MCC Panel Blending_DB"."P-13.02".QRUN;
END_REGION

REGION Network 23: CIP to T-13.00
   RUNG wire#powerrail
      Contact( "AlwaysTRUE" )
      wire#w1
      I_Contact( "General_DB"."Bypass CIP Signal Homomixer" )
      Contact( "CIP_to_Mix".CIP_RequestOK.Homomixer."T-13.00_CIP_RequestOK" )
      wire#w2
      Coil( "T-13.00_Homomixer"."CIP Request OK" )
   END_RUNG
   RUNG wire#w1
      Contact( "General_DB"."Bypass CIP Signal Homomixer" )
   END_RUNG wire#w2
   RUNG wire#w1
      I_Contact( "General_DB"."Bypass CIP Signal Homomixer" )
      Contact( "CIP_to_Mix".CIP_InProgress.Homomixer."T-13.00_CIP_InProgress" )
      wire#w3
      Coil( "T-13.00_Homomixer"."CIP In Progress" )
   END_RUNG
   RUNG wire#w1
      Contact( "General_DB"."Bypass CIP Signal Homomixer" )
   END_RUNG wire#w3
   RUNG wire#w1
      I_Contact( "General_DB"."Bypass CIP Signal Homomixer" )
      Contact( "CIP_to_Mix".CIP_Supply_On.Homomixer."T-13.00_CIP_Supply_ON" )
      wire#w4
      Coil( "T-13.00_Homomixer"."CIP Supply ON" )
   END_RUNG
   RUNG wire#w1
      Contact( "General_DB"."Bypass CIP Signal Homomixer" )
   END_RUNG wire#w4
   RUNG wire#w1
      I_Contact( "General_DB"."Bypass CIP Signal Homomixer" )
      Contact( "CIP_to_Mix".CIP_Complete.Homomixer."T-13.00_CIP_Complete" )
      Coil( "T-13.00_Homomixer"."CIP Complete" )
   END_RUNG
   // the same network as SCL:
   "T-13.00_Homomixer"."CIP Request OK" := "AlwaysTRUE" AND ((NOT "General_DB"."Bypass CIP Signal Homomixer" AND "CIP_to_Mix".CIP_RequestOK.Homomixer."T-13.00_CIP_RequestOK") OR "General_DB"."Bypass CIP Signal Homomixer");
   "T-13.00_Homomixer"."CIP In Progress" := "AlwaysTRUE" AND ((NOT "General_DB"."Bypass CIP Signal Homomixer" AND "CIP_to_Mix".CIP_InProgress.Homomixer."T-13.00_CIP_InProgress") OR "General_DB"."Bypass CIP Signal Homomixer");
   "T-13.00_Homomixer"."CIP Supply ON" := "AlwaysTRUE" AND ((NOT "General_DB"."Bypass CIP Signal Homomixer" AND "CIP_to_Mix".CIP_Supply_On.Homomixer."T-13.00_CIP_Supply_ON") OR "General_DB"."Bypass CIP Signal Homomixer");
   "T-13.00_Homomixer"."CIP Complete" := "AlwaysTRUE" AND NOT "General_DB"."Bypass CIP Signal Homomixer" AND "CIP_to_Mix".CIP_Complete.Homomixer."T-13.00_CIP_Complete";
END_REGION

REGION Network 26: T-14.00 DOSE ON OFF
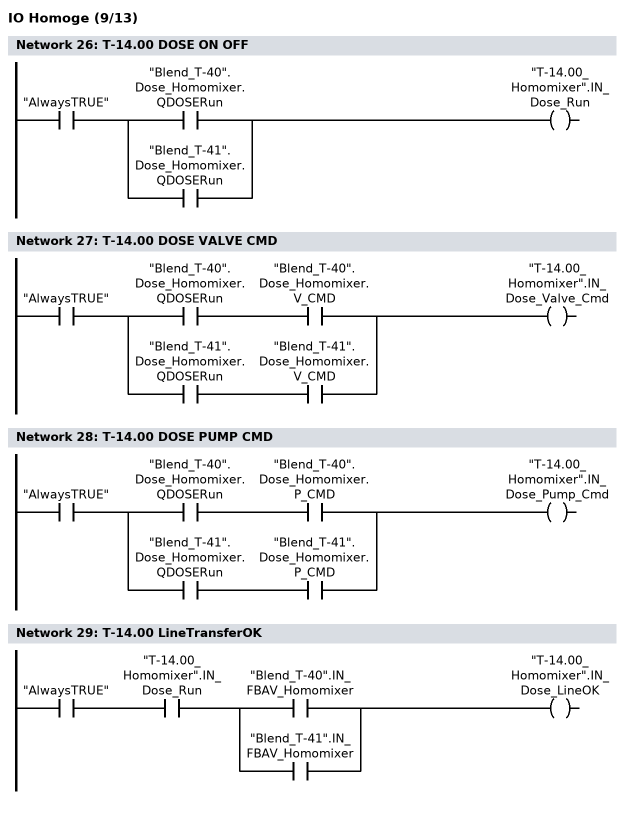
   RUNG wire#powerrail
      Contact( "AlwaysTRUE" )
      wire#w1
      Contact( "Blend_T-40".Dose_Homomixer.QDOSERun )
      wire#w2
      Coil( "T-14.00_Homomixer".IN_Dose_Run )
   END_RUNG
   RUNG wire#w1
      Contact( "Blend_T-41".Dose_Homomixer.QDOSERun )
   END_RUNG wire#w2
   // the same network as SCL:
   "T-14.00_Homomixer".IN_Dose_Run := "AlwaysTRUE" AND ("Blend_T-40".Dose_Homomixer.QDOSERun OR "Blend_T-41".Dose_Homomixer.QDOSERun);
END_REGION

REGION Network 27: T-14.00 DOSE VALVE CMD
   RUNG wire#powerrail
      Contact( "AlwaysTRUE" )
      wire#w1
      Contact( "Blend_T-40".Dose_Homomixer.QDOSERun )
      Contact( "Blend_T-40".Dose_Homomixer.V_CMD )
      wire#w2
      Coil( "T-14.00_Homomixer".IN_Dose_Valve_Cmd )
   END_RUNG
   RUNG wire#w1
      Contact( "Blend_T-41".Dose_Homomixer.QDOSERun )
      Contact( "Blend_T-41".Dose_Homomixer.V_CMD )
   END_RUNG wire#w2
   // the same network as SCL:
   "T-14.00_Homomixer".IN_Dose_Valve_Cmd := "AlwaysTRUE" AND (("Blend_T-40".Dose_Homomixer.QDOSERun AND "Blend_T-40".Dose_Homomixer.V_CMD) OR ("Blend_T-41".Dose_Homomixer.QDOSERun AND "Blend_T-41".Dose_Homomixer.V_CMD));
END_REGION

REGION Network 28: T-14.00 DOSE PUMP CMD
   RUNG wire#powerrail
      Contact( "AlwaysTRUE" )
      wire#w1
      Contact( "Blend_T-40".Dose_Homomixer.QDOSERun )
      Contact( "Blend_T-40".Dose_Homomixer.P_CMD )
      wire#w2
      Coil( "T-14.00_Homomixer".IN_Dose_Pump_Cmd )
   END_RUNG
   RUNG wire#w1
      Contact( "Blend_T-41".Dose_Homomixer.QDOSERun )
      Contact( "Blend_T-41".Dose_Homomixer.P_CMD )
   END_RUNG wire#w2
   // the same network as SCL:
   "T-14.00_Homomixer".IN_Dose_Pump_Cmd := "AlwaysTRUE" AND (("Blend_T-40".Dose_Homomixer.QDOSERun AND "Blend_T-40".Dose_Homomixer.P_CMD) OR ("Blend_T-41".Dose_Homomixer.QDOSERun AND "Blend_T-41".Dose_Homomixer.P_CMD));
END_REGION

REGION Network 29: T-14.00 LineTransferOK
   RUNG wire#powerrail
      Contact( "AlwaysTRUE" )
      Contact( "T-14.00_Homomixer".IN_Dose_Run )
      wire#w1
      Contact( "Blend_T-40".IN_FBAV_Homomixer )
      wire#w2
      Coil( "T-14.00_Homomixer".IN_Dose_LineOK )
   END_RUNG
   RUNG wire#w1
      Contact( "Blend_T-41".IN_FBAV_Homomixer )
   END_RUNG wire#w2
   // the same network as SCL:
   "T-14.00_Homomixer".IN_Dose_LineOK := "AlwaysTRUE" AND "T-14.00_Homomixer".IN_Dose_Run AND ("Blend_T-40".IN_FBAV_Homomixer OR "Blend_T-41".IN_FBAV_Homomixer);
END_REGION

REGION Network 30: T-14.00 Homomixer
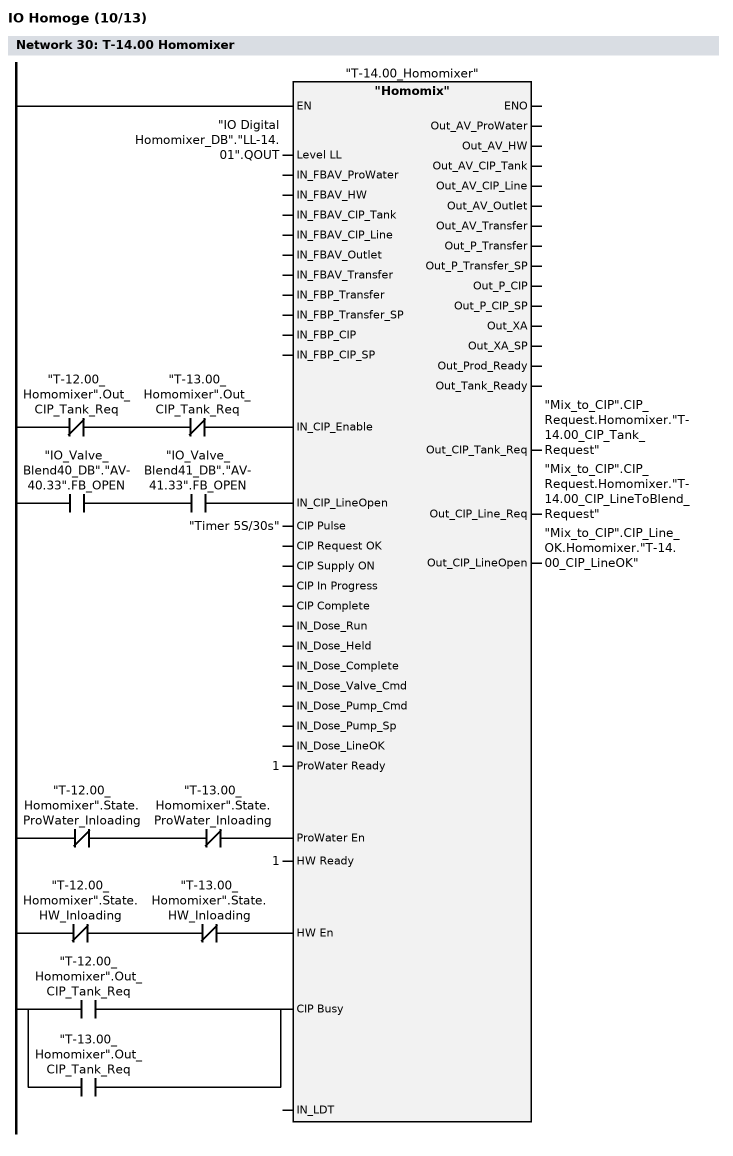
   RUNG wire#powerrail
      "T-14.00_Homomixer"(IN_CIP_Enable := wire#w1, IN_CIP_LineOpen := wire#w2, "ProWater En" := wire#w3, "HW En" := wire#w4, "CIP Busy" := wire#w5, "Level LL" := "IO Digital Homomixer_DB"."LL-14.01".QOUT, IN_FBAV_ProWater :=, IN_FBAV_HW :=, IN_FBAV_CIP_Tank :=, IN_FBAV_CIP_Line :=, IN_FBAV_Outlet :=, IN_FBAV_Transfer :=, IN_FBP_Transfer :=, IN_FBP_Transfer_SP :=, IN_FBP_CIP :=, IN_FBP_CIP_SP :=, "CIP Pulse" := "Timer 5S/30s", "CIP Request OK" :=, "CIP Supply ON" :=, "CIP In Progress" :=, "CIP Complete" :=, IN_Dose_Run :=, IN_Dose_Held :=, IN_Dose_Complete :=, IN_Dose_Valve_Cmd :=, IN_Dose_Pump_Cmd :=, IN_Dose_Pump_Sp :=, IN_Dose_LineOK :=, "ProWater Ready" := 1, "HW Ready" := 1, IN_LDT :=, Out_AV_ProWater =>, Out_AV_HW =>, Out_AV_CIP_Tank =>, Out_AV_CIP_Line =>, Out_AV_Outlet =>, Out_AV_Transfer =>, Out_P_Transfer =>, Out_P_Transfer_SP =>, Out_P_CIP =>, Out_P_CIP_SP =>, Out_XA =>, Out_XA_SP =>, Out_Prod_Ready =>, Out_Tank_Ready =>, Out_CIP_Tank_Req => "Mix_to_CIP".CIP_Request.Homomixer."T-14.00_CIP_Tank_Request", Out_CIP_Line_Req => "Mix_to_CIP".CIP_Request.Homomixer."T-14.00_CIP_LineToBlend_Request", Out_CIP_LineOpen => "Mix_to_CIP".CIP_Line_OK.Homomixer."T-14.00_CIP_LineOK")
   END_RUNG
   RUNG wire#powerrail
      I_Contact( "T-12.00_Homomixer".Out_CIP_Tank_Req )
      I_Contact( "T-13.00_Homomixer".Out_CIP_Tank_Req )
   END_RUNG wire#w1
   RUNG wire#powerrail
      Contact( "IO_Valve_Blend40_DB"."AV-40.33".FB_OPEN )
      Contact( "IO_Valve_Blend41_DB"."AV-41.33".FB_OPEN )
   END_RUNG wire#w2
   RUNG wire#powerrail
      I_Contact( "T-12.00_Homomixer".State.ProWater_Inloading )
      I_Contact( "T-13.00_Homomixer".State.ProWater_Inloading )
   END_RUNG wire#w3
   RUNG wire#powerrail
      I_Contact( "T-12.00_Homomixer".State.HW_Inloading )
      I_Contact( "T-13.00_Homomixer".State.HW_Inloading )
   END_RUNG wire#w4
   RUNG wire#powerrail
      Contact( "T-12.00_Homomixer".Out_CIP_Tank_Req )
   END_RUNG wire#w5
   RUNG wire#powerrail
      Contact( "T-13.00_Homomixer".Out_CIP_Tank_Req )
   END_RUNG wire#w5
   // the same network as SCL:
   "T-14.00_Homomixer"("Level LL" := "IO Digital Homomixer_DB"."LL-14.01".QOUT,   // "Homomix"
                       IN_CIP_Enable := NOT "T-12.00_Homomixer".Out_CIP_Tank_Req AND NOT "T-13.00_Homomixer".Out_CIP_Tank_Req,
                       IN_CIP_LineOpen := "IO_Valve_Blend40_DB"."AV-40.33".FB_OPEN AND "IO_Valve_Blend41_DB"."AV-41.33".FB_OPEN,
                       "CIP Pulse" := "Timer 5S/30s",
                       "ProWater Ready" := 1,
                       "ProWater En" := NOT "T-12.00_Homomixer".State.ProWater_Inloading AND NOT "T-13.00_Homomixer".State.ProWater_Inloading,
                       "HW Ready" := 1,
                       "HW En" := NOT "T-12.00_Homomixer".State.HW_Inloading AND NOT "T-13.00_Homomixer".State.HW_Inloading,
                       "CIP Busy" := "T-12.00_Homomixer".Out_CIP_Tank_Req OR "T-13.00_Homomixer".Out_CIP_Tank_Req,
                       Out_CIP_Tank_Req => "Mix_to_CIP".CIP_Request.Homomixer."T-14.00_CIP_Tank_Request",
                       Out_CIP_Line_Req => "Mix_to_CIP".CIP_Request.Homomixer."T-14.00_CIP_LineToBlend_Request",
                       Out_CIP_LineOpen => "Mix_to_CIP".CIP_Line_OK.Homomixer."T-14.00_CIP_LineOK");
END_REGION

REGION Network 31: T-14.00 Valve Cmd
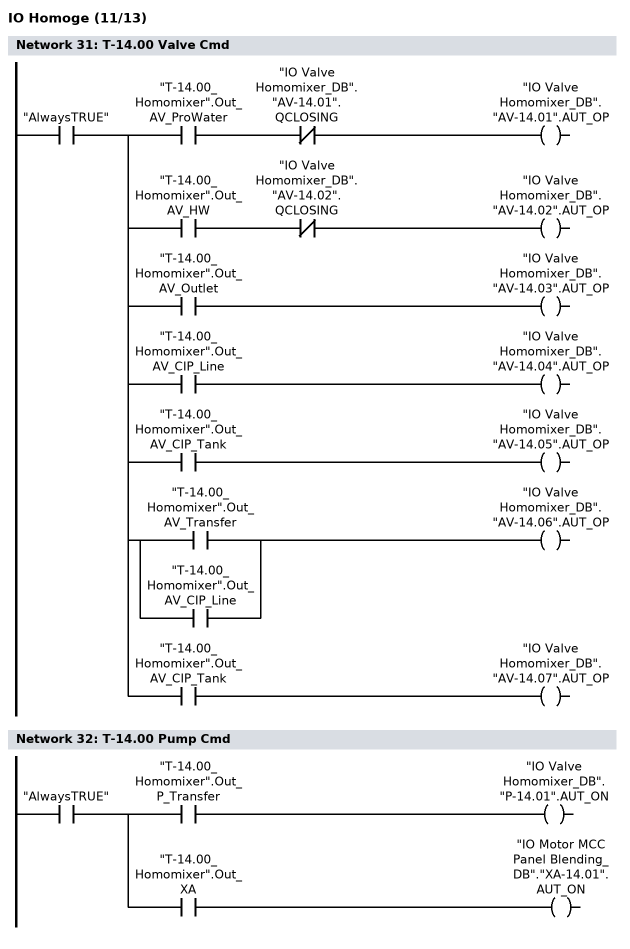
   RUNG wire#powerrail
      Contact( "AlwaysTRUE" )
      wire#w1
      Contact( "T-14.00_Homomixer".Out_AV_ProWater )
      I_Contact( "IO Valve Homomixer_DB"."AV-14.01".QCLOSING )
      Coil( "IO Valve Homomixer_DB"."AV-14.01".AUT_OP )
   END_RUNG
   RUNG wire#w1
      Contact( "T-14.00_Homomixer".Out_AV_HW )
      I_Contact( "IO Valve Homomixer_DB"."AV-14.02".QCLOSING )
      Coil( "IO Valve Homomixer_DB"."AV-14.02".AUT_OP )
   END_RUNG
   RUNG wire#w1
      Contact( "T-14.00_Homomixer".Out_AV_Outlet )
      Coil( "IO Valve Homomixer_DB"."AV-14.03".AUT_OP )
   END_RUNG
   RUNG wire#w1
      Contact( "T-14.00_Homomixer".Out_AV_CIP_Line )
      Coil( "IO Valve Homomixer_DB"."AV-14.04".AUT_OP )
   END_RUNG
   RUNG wire#w1
      Contact( "T-14.00_Homomixer".Out_AV_CIP_Tank )
      Coil( "IO Valve Homomixer_DB"."AV-14.05".AUT_OP )
   END_RUNG
   RUNG wire#w1
      Contact( "T-14.00_Homomixer".Out_AV_Transfer )
      wire#w2
      Coil( "IO Valve Homomixer_DB"."AV-14.06".AUT_OP )
   END_RUNG
   RUNG wire#w1
      Contact( "T-14.00_Homomixer".Out_AV_CIP_Line )
   END_RUNG wire#w2
   RUNG wire#w1
      Contact( "T-14.00_Homomixer".Out_AV_CIP_Tank )
      Coil( "IO Valve Homomixer_DB"."AV-14.07".AUT_OP )
   END_RUNG
   // the same network as SCL:
   "IO Valve Homomixer_DB"."AV-14.01".AUT_OP := "AlwaysTRUE" AND "T-14.00_Homomixer".Out_AV_ProWater AND NOT "IO Valve Homomixer_DB"."AV-14.01".QCLOSING;
   "IO Valve Homomixer_DB"."AV-14.02".AUT_OP := "AlwaysTRUE" AND "T-14.00_Homomixer".Out_AV_HW AND NOT "IO Valve Homomixer_DB"."AV-14.02".QCLOSING;
   "IO Valve Homomixer_DB"."AV-14.03".AUT_OP := "AlwaysTRUE" AND "T-14.00_Homomixer".Out_AV_Outlet;
   "IO Valve Homomixer_DB"."AV-14.04".AUT_OP := "AlwaysTRUE" AND "T-14.00_Homomixer".Out_AV_CIP_Line;
   "IO Valve Homomixer_DB"."AV-14.05".AUT_OP := "AlwaysTRUE" AND "T-14.00_Homomixer".Out_AV_CIP_Tank;
   "IO Valve Homomixer_DB"."AV-14.06".AUT_OP := "AlwaysTRUE" AND ("T-14.00_Homomixer".Out_AV_Transfer OR "T-14.00_Homomixer".Out_AV_CIP_Line);
   "IO Valve Homomixer_DB"."AV-14.07".AUT_OP := "AlwaysTRUE" AND "T-14.00_Homomixer".Out_AV_CIP_Tank;
END_REGION

REGION Network 32: T-14.00 Pump Cmd
   RUNG wire#powerrail
      Contact( "AlwaysTRUE" )
      wire#w1
      Contact( "T-14.00_Homomixer".Out_P_Transfer )
      Coil( "IO Valve Homomixer_DB"."P-14.01".AUT_ON )
   END_RUNG
   RUNG wire#w1
      Contact( "T-14.00_Homomixer".Out_XA )
      Coil( "IO Motor MCC Panel Blending_DB"."XA-14.01".AUT_ON )
   END_RUNG
   // the same network as SCL:
   "IO Valve Homomixer_DB"."P-14.01".AUT_ON := "AlwaysTRUE" AND "T-14.00_Homomixer".Out_P_Transfer;
   "IO Motor MCC Panel Blending_DB"."XA-14.01".AUT_ON := "AlwaysTRUE" AND "T-14.00_Homomixer".Out_XA;
END_REGION

REGION Network 33: T-14.00 Feedback Instrument
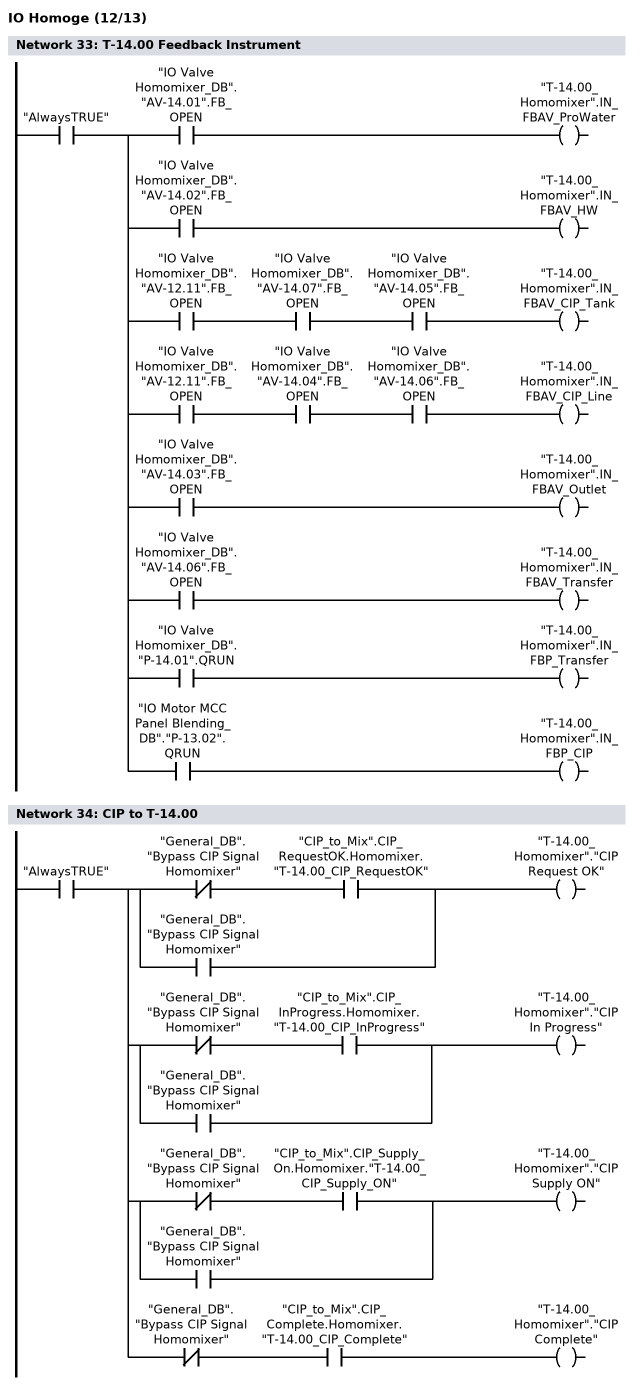
   RUNG wire#powerrail
      Contact( "AlwaysTRUE" )
      wire#w1
      Contact( "IO Valve Homomixer_DB"."AV-14.01".FB_OPEN )
      Coil( "T-14.00_Homomixer".IN_FBAV_ProWater )
   END_RUNG
   RUNG wire#w1
      Contact( "IO Valve Homomixer_DB"."AV-14.02".FB_OPEN )
      Coil( "T-14.00_Homomixer".IN_FBAV_HW )
   END_RUNG
   RUNG wire#w1
      Contact( "IO Valve Homomixer_DB"."AV-12.11".FB_OPEN )
      Contact( "IO Valve Homomixer_DB"."AV-14.07".FB_OPEN )
      Contact( "IO Valve Homomixer_DB"."AV-14.05".FB_OPEN )
      Coil( "T-14.00_Homomixer".IN_FBAV_CIP_Tank )
   END_RUNG
   RUNG wire#w1
      Contact( "IO Valve Homomixer_DB"."AV-12.11".FB_OPEN )
      Contact( "IO Valve Homomixer_DB"."AV-14.04".FB_OPEN )
      Contact( "IO Valve Homomixer_DB"."AV-14.06".FB_OPEN )
      Coil( "T-14.00_Homomixer".IN_FBAV_CIP_Line )
   END_RUNG
   RUNG wire#w1
      Contact( "IO Valve Homomixer_DB"."AV-14.03".FB_OPEN )
      Coil( "T-14.00_Homomixer".IN_FBAV_Outlet )
   END_RUNG
   RUNG wire#w1
      Contact( "IO Valve Homomixer_DB"."AV-14.06".FB_OPEN )
      Coil( "T-14.00_Homomixer".IN_FBAV_Transfer )
   END_RUNG
   RUNG wire#w1
      Contact( "IO Valve Homomixer_DB"."P-14.01".QRUN )
      Coil( "T-14.00_Homomixer".IN_FBP_Transfer )
   END_RUNG
   RUNG wire#w1
      Contact( "IO Motor MCC Panel Blending_DB"."P-13.02".QRUN )
      Coil( "T-14.00_Homomixer".IN_FBP_CIP )
   END_RUNG
   // the same network as SCL:
   "T-14.00_Homomixer".IN_FBAV_ProWater := "AlwaysTRUE" AND "IO Valve Homomixer_DB"."AV-14.01".FB_OPEN;
   "T-14.00_Homomixer".IN_FBAV_HW := "AlwaysTRUE" AND "IO Valve Homomixer_DB"."AV-14.02".FB_OPEN;
   "T-14.00_Homomixer".IN_FBAV_CIP_Tank := "AlwaysTRUE" AND "IO Valve Homomixer_DB"."AV-12.11".FB_OPEN AND "IO Valve Homomixer_DB"."AV-14.07".FB_OPEN AND "IO Valve Homomixer_DB"."AV-14.05".FB_OPEN;
   "T-14.00_Homomixer".IN_FBAV_CIP_Line := "AlwaysTRUE" AND "IO Valve Homomixer_DB"."AV-12.11".FB_OPEN AND "IO Valve Homomixer_DB"."AV-14.04".FB_OPEN AND "IO Valve Homomixer_DB"."AV-14.06".FB_OPEN;
   "T-14.00_Homomixer".IN_FBAV_Outlet := "AlwaysTRUE" AND "IO Valve Homomixer_DB"."AV-14.03".FB_OPEN;
   "T-14.00_Homomixer".IN_FBAV_Transfer := "AlwaysTRUE" AND "IO Valve Homomixer_DB"."AV-14.06".FB_OPEN;
   "T-14.00_Homomixer".IN_FBP_Transfer := "AlwaysTRUE" AND "IO Valve Homomixer_DB"."P-14.01".QRUN;
   "T-14.00_Homomixer".IN_FBP_CIP := "AlwaysTRUE" AND "IO Motor MCC Panel Blending_DB"."P-13.02".QRUN;
END_REGION

REGION Network 34: CIP to T-14.00
   RUNG wire#powerrail
      Contact( "AlwaysTRUE" )
      wire#w1
      I_Contact( "General_DB"."Bypass CIP Signal Homomixer" )
      Contact( "CIP_to_Mix".CIP_RequestOK.Homomixer."T-14.00_CIP_RequestOK" )
      wire#w2
      Coil( "T-14.00_Homomixer"."CIP Request OK" )
   END_RUNG
   RUNG wire#w1
      Contact( "General_DB"."Bypass CIP Signal Homomixer" )
   END_RUNG wire#w2
   RUNG wire#w1
      I_Contact( "General_DB"."Bypass CIP Signal Homomixer" )
      Contact( "CIP_to_Mix".CIP_InProgress.Homomixer."T-14.00_CIP_InProgress" )
      wire#w3
      Coil( "T-14.00_Homomixer"."CIP In Progress" )
   END_RUNG
   RUNG wire#w1
      Contact( "General_DB"."Bypass CIP Signal Homomixer" )
   END_RUNG wire#w3
   RUNG wire#w1
      I_Contact( "General_DB"."Bypass CIP Signal Homomixer" )
      Contact( "CIP_to_Mix".CIP_Supply_On.Homomixer."T-14.00_CIP_Supply_ON" )
      wire#w4
      Coil( "T-14.00_Homomixer"."CIP Supply ON" )
   END_RUNG
   RUNG wire#w1
      Contact( "General_DB"."Bypass CIP Signal Homomixer" )
   END_RUNG wire#w4
   RUNG wire#w1
      I_Contact( "General_DB"."Bypass CIP Signal Homomixer" )
      Contact( "CIP_to_Mix".CIP_Complete.Homomixer."T-14.00_CIP_Complete" )
      Coil( "T-14.00_Homomixer"."CIP Complete" )
   END_RUNG
   // the same network as SCL:
   "T-14.00_Homomixer"."CIP Request OK" := "AlwaysTRUE" AND ((NOT "General_DB"."Bypass CIP Signal Homomixer" AND "CIP_to_Mix".CIP_RequestOK.Homomixer."T-14.00_CIP_RequestOK") OR "General_DB"."Bypass CIP Signal Homomixer");
   "T-14.00_Homomixer"."CIP In Progress" := "AlwaysTRUE" AND ((NOT "General_DB"."Bypass CIP Signal Homomixer" AND "CIP_to_Mix".CIP_InProgress.Homomixer."T-14.00_CIP_InProgress") OR "General_DB"."Bypass CIP Signal Homomixer");
   "T-14.00_Homomixer"."CIP Supply ON" := "AlwaysTRUE" AND ((NOT "General_DB"."Bypass CIP Signal Homomixer" AND "CIP_to_Mix".CIP_Supply_On.Homomixer."T-14.00_CIP_Supply_ON") OR "General_DB"."Bypass CIP Signal Homomixer");
   "T-14.00_Homomixer"."CIP Complete" := "AlwaysTRUE" AND NOT "General_DB"."Bypass CIP Signal Homomixer" AND "CIP_to_Mix".CIP_Complete.Homomixer."T-14.00_CIP_Complete";
END_REGION

REGION Network 36: Valve CIP Supply AV-12.11
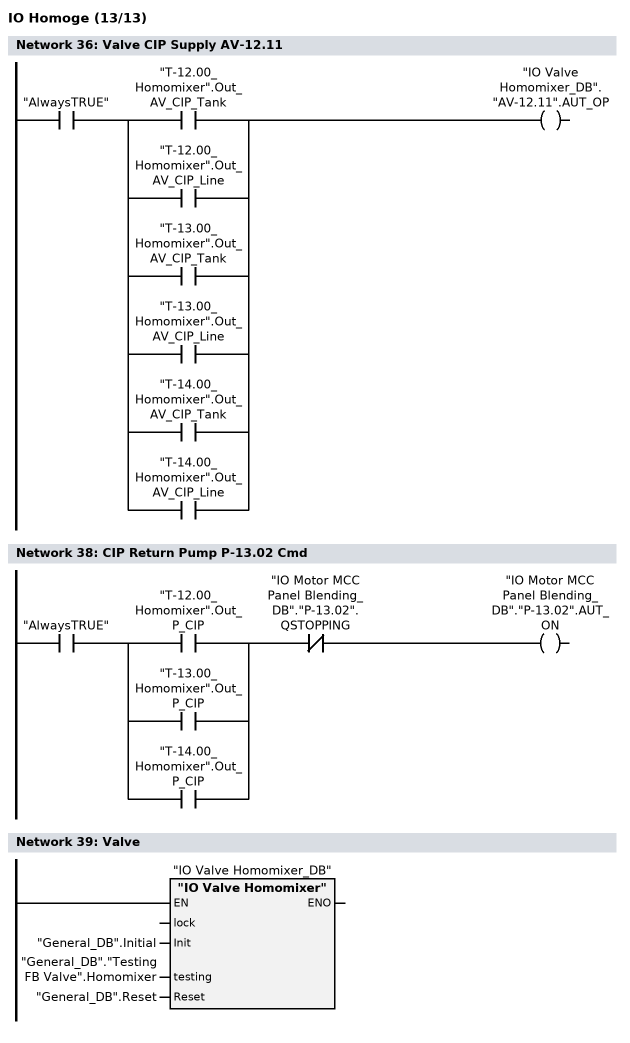
   RUNG wire#powerrail
      Contact( "AlwaysTRUE" )
      wire#w1
      Contact( "T-12.00_Homomixer".Out_AV_CIP_Tank )
      wire#w2
      Coil( "IO Valve Homomixer_DB"."AV-12.11".AUT_OP )
   END_RUNG
   RUNG wire#w1
      Contact( "T-12.00_Homomixer".Out_AV_CIP_Line )
   END_RUNG wire#w2
   RUNG wire#w1
      Contact( "T-13.00_Homomixer".Out_AV_CIP_Tank )
   END_RUNG wire#w2
   RUNG wire#w1
      Contact( "T-13.00_Homomixer".Out_AV_CIP_Line )
   END_RUNG wire#w2
   RUNG wire#w1
      Contact( "T-14.00_Homomixer".Out_AV_CIP_Tank )
   END_RUNG wire#w2
   RUNG wire#w1
      Contact( "T-14.00_Homomixer".Out_AV_CIP_Line )
   END_RUNG wire#w2
   // the same network as SCL:
   "IO Valve Homomixer_DB"."AV-12.11".AUT_OP := "AlwaysTRUE" AND ("T-12.00_Homomixer".Out_AV_CIP_Tank OR "T-12.00_Homomixer".Out_AV_CIP_Line OR "T-13.00_Homomixer".Out_AV_CIP_Tank OR "T-13.00_Homomixer".Out_AV_CIP_Line OR "T-14.00_Homomixer".Out_AV_CIP_Tank OR "T-14.00_Homomixer".Out_AV_CIP_Line);
END_REGION

REGION Network 37: Valve Drain AV-12.12 for T-12 T-13 T-14
END_REGION

REGION Network 38: CIP Return Pump P-13.02 Cmd
   RUNG wire#powerrail
      Contact( "AlwaysTRUE" )
      wire#w1
      Contact( "T-12.00_Homomixer".Out_P_CIP )
      wire#w2
      I_Contact( "IO Motor MCC Panel Blending_DB"."P-13.02".QSTOPPING )
      Coil( "IO Motor MCC Panel Blending_DB"."P-13.02".AUT_ON )
   END_RUNG
   RUNG wire#w1
      Contact( "T-13.00_Homomixer".Out_P_CIP )
   END_RUNG wire#w2
   RUNG wire#w1
      Contact( "T-14.00_Homomixer".Out_P_CIP )
   END_RUNG wire#w2
   // the same network as SCL:
   "IO Motor MCC Panel Blending_DB"."P-13.02".AUT_ON := "AlwaysTRUE" AND ("T-12.00_Homomixer".Out_P_CIP OR "T-13.00_Homomixer".Out_P_CIP OR "T-14.00_Homomixer".Out_P_CIP) AND NOT "IO Motor MCC Panel Blending_DB"."P-13.02".QSTOPPING;
END_REGION

REGION Network 39: Valve
   RUNG wire#powerrail
      "IO Valve Homomixer_DB"(lock :=, Init := "General_DB".Initial, testing := "General_DB"."Testing FB Valve".Homomixer, Reset := "General_DB".Reset)
   END_RUNG
   // the same network as SCL:
   "IO Valve Homomixer_DB"(Init := "General_DB".Initial,   // "IO Valve Homomixer"
                           testing := "General_DB"."Testing FB Valve".Homomixer,
                           Reset := "General_DB".Reset);
END_REGION
END_FUNCTION

FUNCTION_BLOCK "IO Analog Homomixer"   // FB9, LAD
{ S7_Optimized_Access := 'FALSE' }
VERSION : 0.1
// stored: AutoNumber true, IsIECCheckEnabled false, SetENOAutomatically false, UDAEnableTagReadback false
   VAR_INPUT
      Init : Bool;
      Reset : Bool;
   END_VAR
   VAR
      "FT-12.01" : "Ana_w_K1K2";
      "FT-12.02" { S7_SetPoint := 'True'} : "Ana_w_K1K2";
   END_VAR
BEGIN

REGION Network 1: FT-12.01 Flowrate
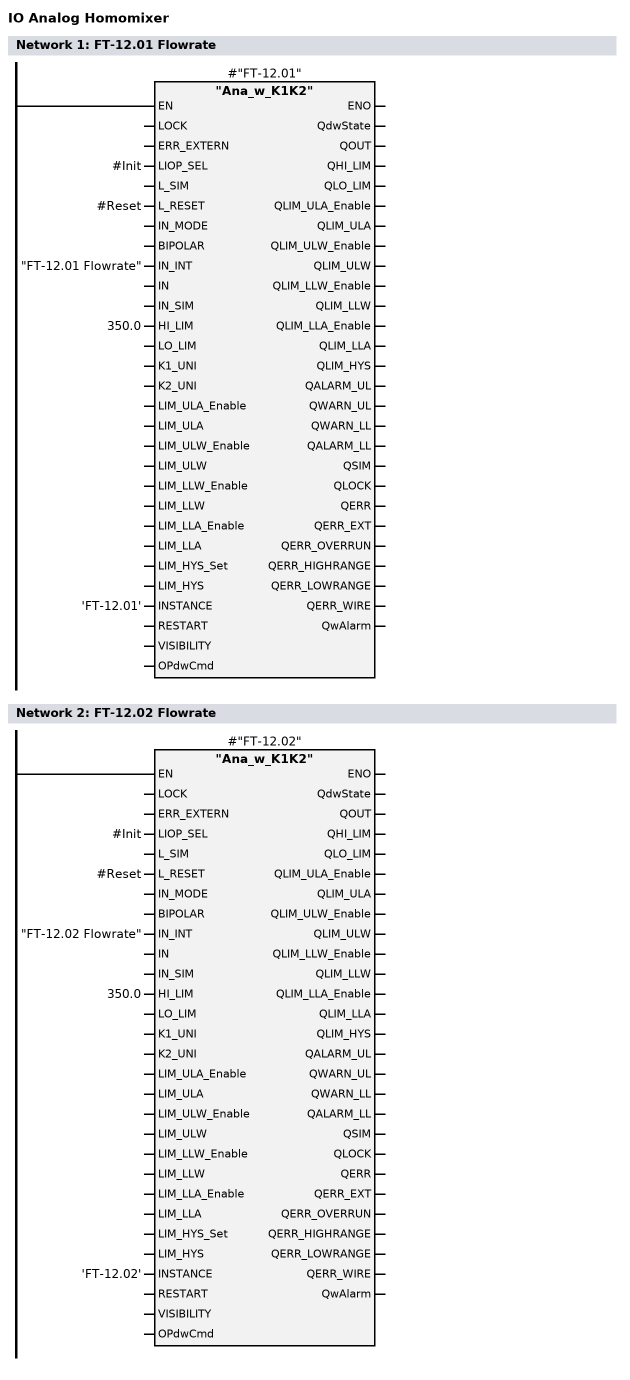
   RUNG wire#powerrail
      #"FT-12.01"(LOCK :=, ERR_EXTERN :=, LIOP_SEL := #Init, L_SIM :=, L_RESET := #Reset, IN_MODE :=, BIPOLAR :=, IN_INT := "FT-12.01 Flowrate", IN :=, IN_SIM :=, HI_LIM := 350.0, LO_LIM :=, K1_UNI :=, K2_UNI :=, LIM_ULA_Enable :=, LIM_ULA :=, LIM_ULW_Enable :=, LIM_ULW :=, LIM_LLW_Enable :=, LIM_LLW :=, LIM_LLA_Enable :=, LIM_LLA :=, LIM_HYS_Set :=, LIM_HYS :=, INSTANCE := 'FT-12.01', RESTART :=, VISIBILITY :=, OPdwCmd :=, QdwState =>, QOUT =>, QHI_LIM =>, QLO_LIM =>, QLIM_ULA_Enable =>, QLIM_ULA =>, QLIM_ULW_Enable =>, QLIM_ULW =>, QLIM_LLW_Enable =>, QLIM_LLW =>, QLIM_LLA_Enable =>, QLIM_LLA =>, QLIM_HYS =>, QALARM_UL =>, QWARN_UL =>, QWARN_LL =>, QALARM_LL =>, QSIM =>, QLOCK =>, QERR =>, QERR_EXT =>, QERR_OVERRUN =>, QERR_HIGHRANGE =>, QERR_LOWRANGE =>, QERR_WIRE =>, QwAlarm =>)
   END_RUNG
   // the same network as SCL:
   #"FT-12.01"(LIOP_SEL := #Init,   // "Ana_w_K1K2"
               L_RESET := #Reset,
               IN_INT := "FT-12.01 Flowrate",
               HI_LIM := 350.0,
               INSTANCE := 'FT-12.01');
END_REGION

REGION Network 2: FT-12.02 Flowrate
   RUNG wire#powerrail
      #"FT-12.02"(LOCK :=, ERR_EXTERN :=, LIOP_SEL := #Init, L_SIM :=, L_RESET := #Reset, IN_MODE :=, BIPOLAR :=, IN_INT := "FT-12.02 Flowrate", IN :=, IN_SIM :=, HI_LIM := 350.0, LO_LIM :=, K1_UNI :=, K2_UNI :=, LIM_ULA_Enable :=, LIM_ULA :=, LIM_ULW_Enable :=, LIM_ULW :=, LIM_LLW_Enable :=, LIM_LLW :=, LIM_LLA_Enable :=, LIM_LLA :=, LIM_HYS_Set :=, LIM_HYS :=, INSTANCE := 'FT-12.02', RESTART :=, VISIBILITY :=, OPdwCmd :=, QdwState =>, QOUT =>, QHI_LIM =>, QLO_LIM =>, QLIM_ULA_Enable =>, QLIM_ULA =>, QLIM_ULW_Enable =>, QLIM_ULW =>, QLIM_LLW_Enable =>, QLIM_LLW =>, QLIM_LLA_Enable =>, QLIM_LLA =>, QLIM_HYS =>, QALARM_UL =>, QWARN_UL =>, QWARN_LL =>, QALARM_LL =>, QSIM =>, QLOCK =>, QERR =>, QERR_EXT =>, QERR_OVERRUN =>, QERR_HIGHRANGE =>, QERR_LOWRANGE =>, QERR_WIRE =>, QwAlarm =>)
   END_RUNG
   // the same network as SCL:
   #"FT-12.02"(LIOP_SEL := #Init,   // "Ana_w_K1K2"
               L_RESET := #Reset,
               IN_INT := "FT-12.02 Flowrate",
               HI_LIM := 350.0,
               INSTANCE := 'FT-12.02');
END_REGION
END_FUNCTION_BLOCK

FUNCTION_BLOCK "IO Digital Homomixer"   // FB5, LAD
{ S7_Optimized_Access := 'FALSE' }
VERSION : 0.1
// stored: AutoNumber true, IsIECCheckEnabled false, SetENOAutomatically false, UDAEnableTagReadback false
   VAR_INPUT
      Init : Bool;
      Reset : Bool;
   END_VAR
   VAR
      "LL-12.01" { S7_SetPoint := 'True'} : "Digital";   // LOW LEVEL SENSOR HOMOMIXER T-12.00
      "LL-13.01" { S7_SetPoint := 'True'} : "Digital";   // LOW LEVEL SENSOR HOMOMIXER T-13.00
      "LL-14.01" { S7_SetPoint := 'True'} : "Digital";
   END_VAR
BEGIN

REGION Network 1: LL-12.01 LOW LEVEL SENSOR HOMOMIXER T-12.00
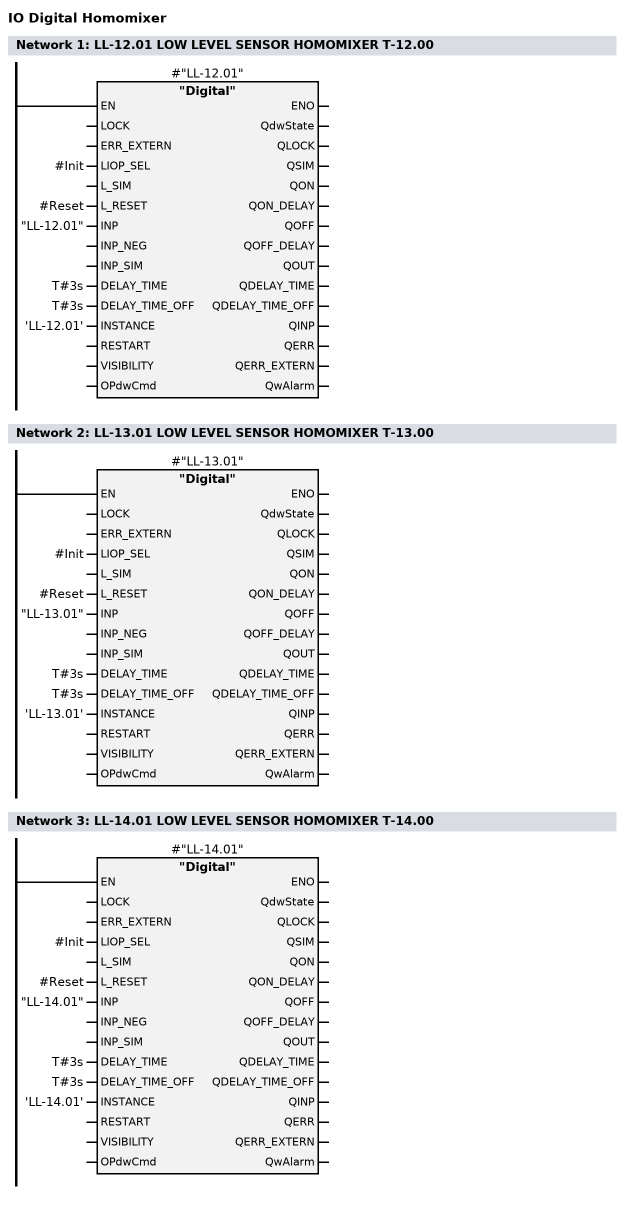
   RUNG wire#powerrail
      #"LL-12.01"(LOCK :=, ERR_EXTERN :=, LIOP_SEL := #Init, L_SIM :=, L_RESET := #Reset, INP := "LL-12.01", INP_NEG :=, INP_SIM :=, DELAY_TIME := T#3s, DELAY_TIME_OFF := T#3s, INSTANCE := 'LL-12.01', RESTART :=, VISIBILITY :=, OPdwCmd :=, QdwState =>, QLOCK =>, QSIM =>, QON =>, QON_DELAY =>, QOFF =>, QOFF_DELAY =>, QOUT =>, QDELAY_TIME =>, QDELAY_TIME_OFF =>, QINP =>, QERR =>, QERR_EXTERN =>, QwAlarm =>)
   END_RUNG
   // the same network as SCL:
   #"LL-12.01"(LIOP_SEL := #Init,   // "Digital"
               L_RESET := #Reset,
               INP := "LL-12.01",
               DELAY_TIME := T#3s,
               DELAY_TIME_OFF := T#3s,
               INSTANCE := 'LL-12.01');
END_REGION

REGION Network 2: LL-13.01 LOW LEVEL SENSOR HOMOMIXER T-13.00
   RUNG wire#powerrail
      #"LL-13.01"(LOCK :=, ERR_EXTERN :=, LIOP_SEL := #Init, L_SIM :=, L_RESET := #Reset, INP := "LL-13.01", INP_NEG :=, INP_SIM :=, DELAY_TIME := T#3s, DELAY_TIME_OFF := T#3s, INSTANCE := 'LL-13.01', RESTART :=, VISIBILITY :=, OPdwCmd :=, QdwState =>, QLOCK =>, QSIM =>, QON =>, QON_DELAY =>, QOFF =>, QOFF_DELAY =>, QOUT =>, QDELAY_TIME =>, QDELAY_TIME_OFF =>, QINP =>, QERR =>, QERR_EXTERN =>, QwAlarm =>)
   END_RUNG
   // the same network as SCL:
   #"LL-13.01"(LIOP_SEL := #Init,   // "Digital"
               L_RESET := #Reset,
               INP := "LL-13.01",
               DELAY_TIME := T#3s,
               DELAY_TIME_OFF := T#3s,
               INSTANCE := 'LL-13.01');
END_REGION

REGION Network 3: LL-14.01 LOW LEVEL SENSOR HOMOMIXER T-14.00
   RUNG wire#powerrail
      #"LL-14.01"(LOCK :=, ERR_EXTERN :=, LIOP_SEL := #Init, L_SIM :=, L_RESET := #Reset, INP := "LL-14.01", INP_NEG :=, INP_SIM :=, DELAY_TIME := T#3s, DELAY_TIME_OFF := T#3s, INSTANCE := 'LL-14.01', RESTART :=, VISIBILITY :=, OPdwCmd :=, QdwState =>, QLOCK =>, QSIM =>, QON =>, QON_DELAY =>, QOFF =>, QOFF_DELAY =>, QOUT =>, QDELAY_TIME =>, QDELAY_TIME_OFF =>, QINP =>, QERR =>, QERR_EXTERN =>, QwAlarm =>)
   END_RUNG
   // the same network as SCL:
   #"LL-14.01"(LIOP_SEL := #Init,   // "Digital"
               L_RESET := #Reset,
               INP := "LL-14.01",
               DELAY_TIME := T#3s,
               DELAY_TIME_OFF := T#3s,
               INSTANCE := 'LL-14.01');
END_REGION
END_FUNCTION_BLOCK

FUNCTION_BLOCK "Homomix"   // FB18, LAD
{ S7_Optimized_Access := 'TRUE' }
VERSION : 0.1
// stored: AutoNumber true, IsIECCheckEnabled false, IsRetainMemResEnabled false, MemoryReserve 100, SetENOAutomatically false, UDAEnableTagReadback false
   VAR_INPUT
      "Level LL" : Bool;
      IN_FBAV_ProWater : Bool;
      IN_FBAV_HW : Bool;
      IN_FBAV_CIP_Tank : Bool;
      IN_FBAV_CIP_Line : Bool;
      IN_FBAV_Outlet : Bool;
      IN_FBAV_Transfer : Bool;
      IN_FBP_Transfer : Bool;
      IN_FBP_Transfer_SP : Real;
      IN_FBP_CIP : Bool;
      IN_FBP_CIP_SP : Real;
      IN_CIP_Enable : Bool;
      IN_CIP_LineOpen : Bool;
      "CIP Pulse" : Bool;
      "CIP Request OK" : Bool;
      "CIP Supply ON" : Bool;
      "CIP In Progress" : Bool;
      "CIP Complete" : Bool;
      IN_Dose_Run : Bool;
      IN_Dose_Held : Bool;
      IN_Dose_Complete : Bool;
      IN_Dose_Valve_Cmd : Bool;
      IN_Dose_Pump_Cmd : Bool;
      IN_Dose_Pump_Sp : Real;
      IN_Dose_LineOK : Bool;
      "ProWater Ready" : Bool;
      "ProWater En" : Bool;
      "HW Ready" : Bool;
      "HW En" : Bool;
      "CIP Busy" : Bool;
      IN_LDT : Date_And_Time;
   END_VAR
   VAR_OUTPUT
      Out_AV_ProWater : Bool;
      Out_AV_HW : Bool;
      Out_AV_CIP_Tank : Bool;
      Out_AV_CIP_Line : Bool;
      Out_AV_Outlet : Bool;
      Out_AV_Transfer : Bool;
      Out_P_Transfer : Bool;
      Out_P_Transfer_SP : Real;
      Out_P_CIP : Bool;
      Out_P_CIP_SP : Real;
      Out_XA : Bool;
      Out_XA_SP : Real;
      Out_Prod_Ready : Bool;
      Out_Tank_Ready : Bool;
      Out_CIP_Tank_Req : Bool;
      Out_CIP_Line_Req : Bool;
      Out_CIP_LineOpen : Bool;
   END_VAR
   VAR
      Cmd : Struct
         Ready_for_Transfer : Bool;
         "CIP Tank" : Bool;
         "CIP Line" : Bool;
         "Agi Mode" : Bool;
         "Agi ON OFF" : Bool;
      END_STRUCT;
   END_VAR
   VAR RETAIN
      Param : Struct
         "CIP Pump SP" : Real := 50.0;
         "Agi SP" : Real := 50.0;
         Dose_HW_SP : Real;
         Dose_ProWater_SP : Real;
         LastDose_HW : Real;
         LastDose_ProWater : Real;
      END_STRUCT;
   END_VAR
   VAR
      State : Struct
         "Tank LL" : Bool;
         "CIP Tank" : Bool;
         "CIP Tank Ena" : Bool;
         "CIP Line" : Bool;
         "CIP Line Ena" : Bool;
         "CIP Return On" : Bool;
         "Dose EN" : Bool;
         ProWater_Inloading : Bool;
         HW_Inloading : Bool;
         Tank_Inloading : Bool;
         "Ready For Transfer" : Bool;
         "Ready For Transfer EN" : Bool;
         Transfer_On_Prog : Bool;
         "CIP Req" : Bool;
      END_STRUCT;
      Dose : Struct
         Dose_Start : DWord;
         Dose_Pause : DWord;
         Dose_Stop : DWord;
         Dose_State : DWord;
         Dose_Tank_Available : Word;
         Dose_Prod_Ready : Word;
         Dose_Header_Req : DWord;
         Dose_EN : Word;
      END_STRUCT;
      SP_ProWater : "Raw_Pulse";
      SP_HW { S7_SetPoint := 'True'} : "Raw_Pulse";
      Dose_ProWater { S7_SetPoint := 'True'} : "DOSE";
      Dose_HW { S7_SetPoint := 'True'} : "DOSE";
      r : Struct
         PosE1 : Bool;
         PosE2 : Bool;
         PosE3 : Bool;
         PosE4 : Bool;
         PosE5 : Bool;
         PosE6 : Bool;
         PosE7 : Bool;
         PosE8 : Bool;
         PosE9 : Bool;
         PosE10 : Bool;
         PosE11 : Bool;
         PosE12 : Bool;
         PosE13 : Bool;
         PosE14 : Bool;
         PosE15 : Bool;
         PosE16 : Bool;
         PosE17 : Bool;
         PosE18 : Bool;
         PosE19 : Bool;
         PosE20 : Bool;
         PosE21 : Bool;
         PosE22 : Bool;
         PosE23 : Bool;
         PosE24 : Bool;
         PosE25 : Bool;
         PosE26 : Bool;
         PosE27 : Bool;
         PosE28 : Bool;
         PosE29 : Bool;
         PosE30 : Bool;
         PosE31 : Bool;
         PosE32 : Bool;
      END_STRUCT;
      CIPRetOn_Time : TON_TIME;
      CIPRetOff_Time { S7_SetPoint := 'True'} : TON_TIME;
      Actuator : Struct
         AV_Transfer : Bool;
         AV_Outlet : Bool;
         AV_CIP : Bool;
         P_Transfer : Bool;
         P_CIP : Bool;
      END_STRUCT;
      alwaysOn : Bool;
   END_VAR
   VAR RETAIN
      TimerON : Struct
         TimerON_1 : TON_TIME;
         TimerON_2 { S7_SetPoint := 'True'} : TON_TIME;
         TimerON_3 { S7_SetPoint := 'True'} : TON_TIME;
         TimerON_4 { S7_SetPoint := 'True'} : TON_TIME;
         TimerON_5 { S7_SetPoint := 'True'} : TON_TIME;
         TimerON_6 { S7_SetPoint := 'True'} : TON_TIME;
         TimerON_7 { S7_SetPoint := 'True'} : TON_TIME;
         TimerON_8 { S7_SetPoint := 'True'} : TON_TIME;
      END_STRUCT;
   END_VAR
   VAR_TEMP
      b_transfer : Bool;
   END_VAR
   // SP_ProWater.Para."SP_Qty_Fine%" := 10.0;
   // SP_HW.Para."SP_Qty_Fine%" := 10.0;
   // TimerON.TimerON_1.PT := T#10s;
   // TimerON.TimerON_2.PT := T#10s;
   // TimerON.TimerON_3.PT := T#10s;
   // TimerON.TimerON_4.PT := T#10s;
   // TimerON.TimerON_5.PT := T#10s;
   // TimerON.TimerON_6.PT := T#10s;
   // TimerON.TimerON_7.PT := T#10s;
   // TimerON.TimerON_8.PT := T#10s;
   VAR_TEMP   // added for the SCL form of the ladder/FBD networks
      _w1 : Bool;
      _w2 : Bool;
   END_VAR
BEGIN

REGION Network 1: Always ON
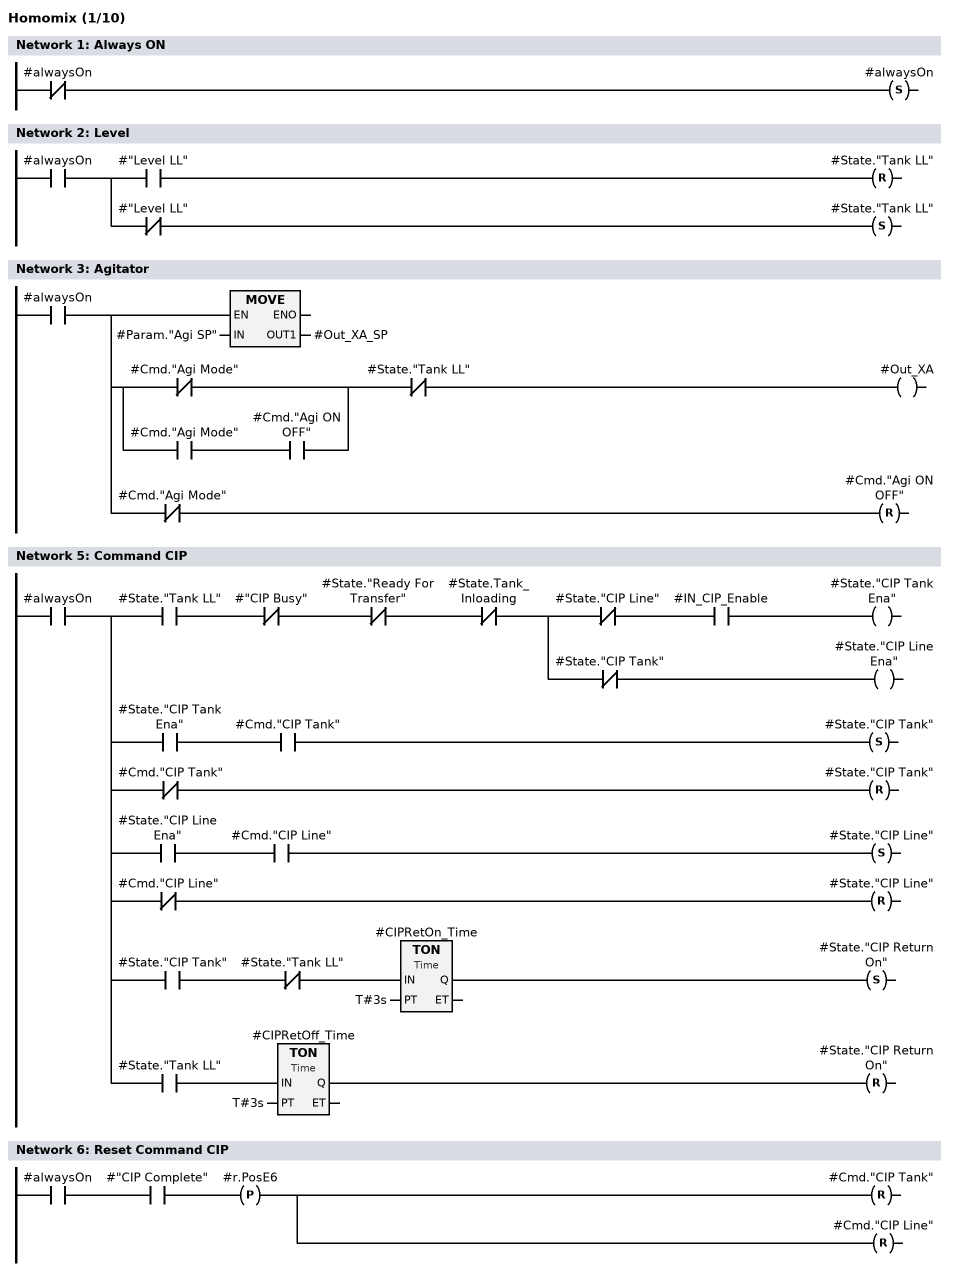
   RUNG wire#powerrail
      I_Contact( #alwaysOn )
      S_Coil( #alwaysOn )
   END_RUNG
   // the same network as SCL:
   IF NOT #alwaysOn THEN #alwaysOn := TRUE; END_IF;
END_REGION

REGION Network 2: Level
   RUNG wire#powerrail
      Contact( #alwaysOn )
      wire#w1
      Contact( #"Level LL" )
      R_Coil( #State."Tank LL" )
   END_RUNG
   RUNG wire#w1
      I_Contact( #"Level LL" )
      S_Coil( #State."Tank LL" )
   END_RUNG
   // the same network as SCL:
   IF #alwaysOn AND #"Level LL" THEN #State."Tank LL" := FALSE; END_IF;
   IF #alwaysOn AND NOT #"Level LL" THEN #State."Tank LL" := TRUE; END_IF;
END_REGION

REGION Network 3: Agitator
   RUNG wire#powerrail
      Contact( #alwaysOn )
      wire#w1
      Move(in := #Param."Agi SP", out1 => #Out_XA_SP)
   END_RUNG
   RUNG wire#w1
      I_Contact( #Cmd."Agi Mode" )
      wire#w2
      I_Contact( #State."Tank LL" )
      Coil( #Out_XA )
   END_RUNG
   RUNG wire#w1
      Contact( #Cmd."Agi Mode" )
      Contact( #Cmd."Agi ON OFF" )
   END_RUNG wire#w2
   RUNG wire#w1
      I_Contact( #Cmd."Agi Mode" )
      R_Coil( #Cmd."Agi ON OFF" )
   END_RUNG
   // the same network as SCL:
   IF #alwaysOn THEN #Out_XA_SP := #Param."Agi SP"; END_IF;
   #Out_XA := #alwaysOn AND (NOT #Cmd."Agi Mode" OR (#Cmd."Agi Mode" AND #Cmd."Agi ON OFF")) AND NOT #State."Tank LL";
   IF #alwaysOn AND NOT #Cmd."Agi Mode" THEN #Cmd."Agi ON OFF" := FALSE; END_IF;
END_REGION

REGION Network 5: Command CIP
   RUNG wire#powerrail
      Contact( #alwaysOn )
      wire#w1
      Contact( #State."Tank LL" )
      I_Contact( #"CIP Busy" )
      I_Contact( #State."Ready For Transfer" )
      I_Contact( #State.Tank_Inloading )
      wire#w2
      I_Contact( #State."CIP Line" )
      Contact( #IN_CIP_Enable )
      Coil( #State."CIP Tank Ena" )
   END_RUNG
   RUNG wire#w2
      I_Contact( #State."CIP Tank" )
      Coil( #State."CIP Line Ena" )
   END_RUNG
   RUNG wire#w1
      Contact( #State."CIP Tank Ena" )
      Contact( #Cmd."CIP Tank" )
      S_Coil( #State."CIP Tank" )
   END_RUNG
   RUNG wire#w1
      I_Contact( #Cmd."CIP Tank" )
      R_Coil( #State."CIP Tank" )
   END_RUNG
   RUNG wire#w1
      Contact( #State."CIP Line Ena" )
      Contact( #Cmd."CIP Line" )
      S_Coil( #State."CIP Line" )
   END_RUNG
   RUNG wire#w1
      I_Contact( #Cmd."CIP Line" )
      R_Coil( #State."CIP Line" )
   END_RUNG
   RUNG wire#w1
      Contact( #State."CIP Tank" )
      I_Contact( #State."Tank LL" )
      { S7_Templates := "time_type := Time" } #CIPRetOn_Time.TON(pt := T#3s, et =>)
      S_Coil( #State."CIP Return On" )
   END_RUNG
   RUNG wire#w1
      Contact( #State."Tank LL" )
      { S7_Templates := "time_type := Time" } #CIPRetOff_Time.TON(pt := T#3s, et =>)
      R_Coil( #State."CIP Return On" )
   END_RUNG
   // the same network as SCL:
   #_w1 := #alwaysOn AND #State."Tank LL" AND NOT #"CIP Busy" AND NOT #State."Ready For Transfer" AND NOT #State.Tank_Inloading;
   #State."CIP Tank Ena" := #_w1 AND NOT #State."CIP Line" AND #IN_CIP_Enable;
   #State."CIP Line Ena" := #_w1 AND NOT #State."CIP Tank";
   IF #alwaysOn AND #State."CIP Tank Ena" AND #Cmd."CIP Tank" THEN #State."CIP Tank" := TRUE; END_IF;
   IF #alwaysOn AND NOT #Cmd."CIP Tank" THEN #State."CIP Tank" := FALSE; END_IF;
   IF #alwaysOn AND #State."CIP Line Ena" AND #Cmd."CIP Line" THEN #State."CIP Line" := TRUE; END_IF;
   IF #alwaysOn AND NOT #Cmd."CIP Line" THEN #State."CIP Line" := FALSE; END_IF;
   #CIPRetOn_Time(IN := #alwaysOn AND #State."CIP Tank" AND NOT #State."Tank LL", PT := T#3s);   // TON
   IF #CIPRetOn_Time.Q THEN #State."CIP Return On" := TRUE; END_IF;
   #CIPRetOff_Time(IN := #alwaysOn AND #State."Tank LL", PT := T#3s);   // TON
   IF #CIPRetOff_Time.Q THEN #State."CIP Return On" := FALSE; END_IF;
END_REGION

REGION Network 6: Reset Command CIP
   RUNG wire#powerrail
      Contact( #alwaysOn )
      Contact( #"CIP Complete" )
      P_Trig( #r.PosE6 )
      wire#w1
      R_Coil( #Cmd."CIP Tank" )
   END_RUNG
   RUNG wire#w1
      R_Coil( #Cmd."CIP Line" )
   END_RUNG
   // the same network as SCL:
   #_w1 := #alwaysOn AND #"CIP Complete";
   #_w2 := #_w1 AND NOT #r.PosE6;   // rising edge
   #r.PosE6 := #_w1;
   IF #_w2 THEN
       #Cmd."CIP Tank" := FALSE;
       #Cmd."CIP Line" := FALSE;
   END_IF;
END_REGION

REGION Network 7: CIP Request and CIP Line Open
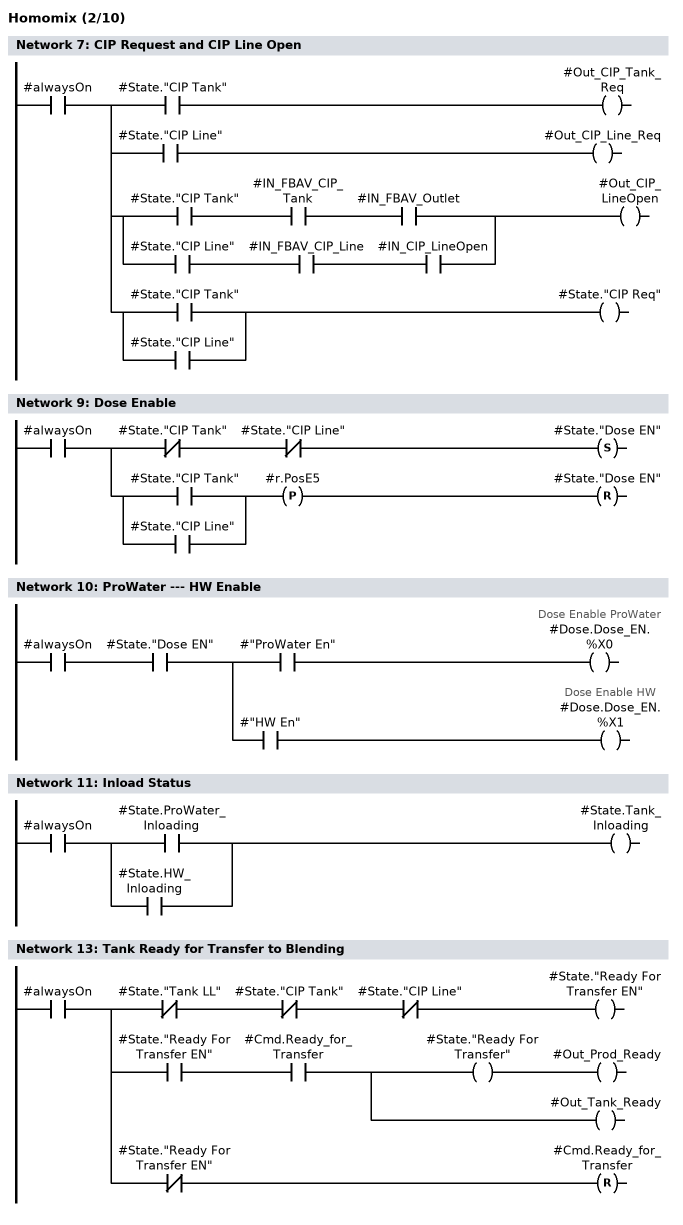
   RUNG wire#powerrail
      Contact( #alwaysOn )
      wire#w1
      Contact( #State."CIP Tank" )
      Coil( #Out_CIP_Tank_Req )
   END_RUNG
   RUNG wire#w1
      Contact( #State."CIP Line" )
      Coil( #Out_CIP_Line_Req )
   END_RUNG
   RUNG wire#w1
      Contact( #State."CIP Tank" )
      Contact( #IN_FBAV_CIP_Tank )
      Contact( #IN_FBAV_Outlet )
      wire#w2
      Coil( #Out_CIP_LineOpen )
   END_RUNG
   RUNG wire#w1
      Contact( #State."CIP Line" )
      Contact( #IN_FBAV_CIP_Line )
      Contact( #IN_CIP_LineOpen )
   END_RUNG wire#w2
   RUNG wire#w1
      Contact( #State."CIP Tank" )
      wire#w3
      Coil( #State."CIP Req" )
   END_RUNG
   RUNG wire#w1
      Contact( #State."CIP Line" )
   END_RUNG wire#w3
   // the same network as SCL:
   #Out_CIP_Tank_Req := #alwaysOn AND #State."CIP Tank";
   #Out_CIP_Line_Req := #alwaysOn AND #State."CIP Line";
   #Out_CIP_LineOpen := #alwaysOn AND ((#State."CIP Tank" AND #IN_FBAV_CIP_Tank AND #IN_FBAV_Outlet) OR (#State."CIP Line" AND #IN_FBAV_CIP_Line AND #IN_CIP_LineOpen));
   #State."CIP Req" := #alwaysOn AND (#State."CIP Tank" OR #State."CIP Line");
END_REGION

REGION Network 9: Dose Enable
   RUNG wire#powerrail
      Contact( #alwaysOn )
      wire#w1
      I_Contact( #State."CIP Tank" )
      I_Contact( #State."CIP Line" )
      S_Coil( #State."Dose EN" )
   END_RUNG
   RUNG wire#w1
      Contact( #State."CIP Tank" )
      wire#w2
      P_Trig( #r.PosE5 )
      R_Coil( #State."Dose EN" )
   END_RUNG
   RUNG wire#w1
      Contact( #State."CIP Line" )
   END_RUNG wire#w2
   // the same network as SCL:
   IF #alwaysOn AND NOT #State."CIP Tank" AND NOT #State."CIP Line" THEN #State."Dose EN" := TRUE; END_IF;
   #_w1 := #alwaysOn AND (#State."CIP Tank" OR #State."CIP Line");
   #_w2 := #_w1 AND NOT #r.PosE5;   // rising edge
   #r.PosE5 := #_w1;
   IF #_w2 THEN #State."Dose EN" := FALSE; END_IF;
END_REGION

REGION Network 10: ProWater --- HW Enable
   RUNG wire#powerrail
      Contact( #alwaysOn )
      Contact( #State."Dose EN" )
      wire#w1
      Contact( #"ProWater En" )
      Coil( #Dose.Dose_EN.%X0 )   // Dose Enable ProWater
   END_RUNG
   RUNG wire#w1
      Contact( #"HW En" )
      Coil( #Dose.Dose_EN.%X1 )   // Dose Enable HW
   END_RUNG
   // the same network as SCL:
   #_w1 := #alwaysOn AND #State."Dose EN";
   #Dose.Dose_EN.%X0 := #_w1 AND #"ProWater En";   // Dose Enable ProWater
   #Dose.Dose_EN.%X1 := #_w1 AND #"HW En";   // Dose Enable HW
END_REGION

REGION Network 11: Inload Status
   RUNG wire#powerrail
      Contact( #alwaysOn )
      wire#w1
      Contact( #State.ProWater_Inloading )
      wire#w2
      Coil( #State.Tank_Inloading )
   END_RUNG
   RUNG wire#w1
      Contact( #State.HW_Inloading )
   END_RUNG wire#w2
   // the same network as SCL:
   #State.Tank_Inloading := #alwaysOn AND (#State.ProWater_Inloading OR #State.HW_Inloading);
END_REGION

REGION Network 13: Tank Ready for Transfer to Blending
   RUNG wire#powerrail
      Contact( #alwaysOn )
      wire#w1
      I_Contact( #State."Tank LL" )
      I_Contact( #State."CIP Tank" )
      I_Contact( #State."CIP Line" )
      Coil( #State."Ready For Transfer EN" )
   END_RUNG
   RUNG wire#w1
      Contact( #State."Ready For Transfer EN" )
      Contact( #Cmd.Ready_for_Transfer )
      wire#w2
      Coil( #State."Ready For Transfer" )
      Coil( #Out_Prod_Ready )
   END_RUNG
   RUNG wire#w2
      Coil( #Out_Tank_Ready )
   END_RUNG
   RUNG wire#w1
      I_Contact( #State."Ready For Transfer EN" )
      R_Coil( #Cmd.Ready_for_Transfer )
   END_RUNG
   // the same network as SCL:
   #State."Ready For Transfer EN" := #alwaysOn AND NOT #State."Tank LL" AND NOT #State."CIP Tank" AND NOT #State."CIP Line";
   #State."Ready For Transfer" := #alwaysOn AND #State."Ready For Transfer EN" AND #Cmd.Ready_for_Transfer;
   #Out_Prod_Ready := #State."Ready For Transfer";
   #Out_Tank_Ready := #State."Ready For Transfer";
   IF #alwaysOn AND NOT #State."Ready For Transfer EN" THEN #Cmd.Ready_for_Transfer := FALSE; END_IF;
END_REGION

REGION Network 14: Transfer to Blending AV and Pump
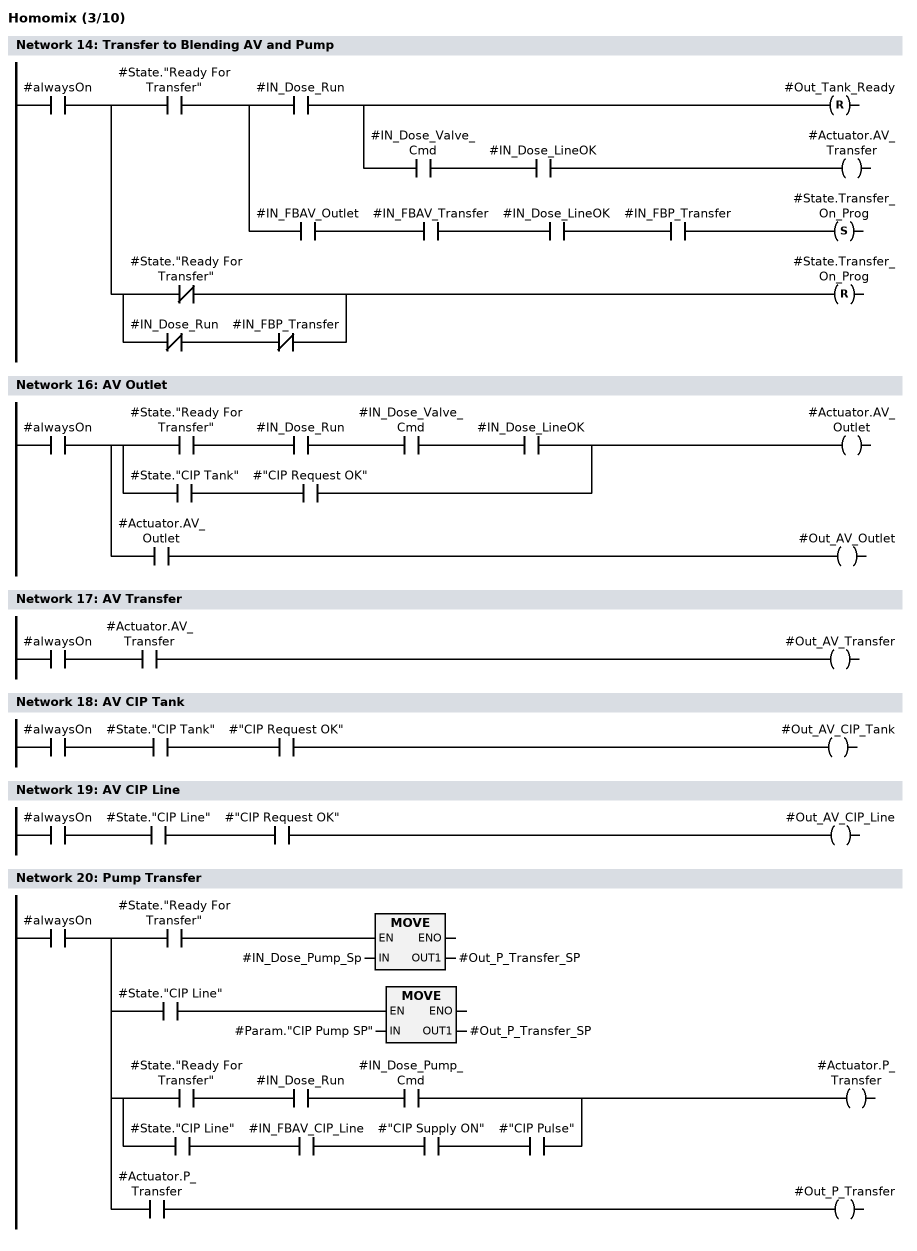
   RUNG wire#powerrail
      Contact( #alwaysOn )
      wire#w1
      Contact( #State."Ready For Transfer" )
      wire#w2
      Contact( #IN_Dose_Run )
      wire#w3
      R_Coil( #Out_Tank_Ready )
   END_RUNG
   RUNG wire#w3
      Contact( #IN_Dose_Valve_Cmd )
      Contact( #IN_Dose_LineOK )
      Coil( #Actuator.AV_Transfer )
   END_RUNG
   RUNG wire#w2
      Contact( #IN_FBAV_Outlet )
      Contact( #IN_FBAV_Transfer )
      Contact( #IN_Dose_LineOK )
      Contact( #IN_FBP_Transfer )
      S_Coil( #State.Transfer_On_Prog )
   END_RUNG
   RUNG wire#w1
      I_Contact( #State."Ready For Transfer" )
      wire#w4
      R_Coil( #State.Transfer_On_Prog )
   END_RUNG
   RUNG wire#w1
      I_Contact( #IN_Dose_Run )
      I_Contact( #IN_FBP_Transfer )
   END_RUNG wire#w4
   // the same network as SCL:
   #_w1 := #alwaysOn AND #State."Ready For Transfer";
   #_w2 := #_w1 AND #IN_Dose_Run;
   IF #_w2 THEN #Out_Tank_Ready := FALSE; END_IF;
   #Actuator.AV_Transfer := #_w2 AND #IN_Dose_Valve_Cmd AND #IN_Dose_LineOK;
   IF #_w1 AND #IN_FBAV_Outlet AND #IN_FBAV_Transfer AND #IN_Dose_LineOK AND #IN_FBP_Transfer THEN
       #State.Transfer_On_Prog := TRUE;
   END_IF;
   IF #alwaysOn AND (NOT #State."Ready For Transfer" OR (NOT #IN_Dose_Run AND NOT #IN_FBP_Transfer)) THEN
       #State.Transfer_On_Prog := FALSE;
   END_IF;
END_REGION

REGION Network 16: AV Outlet
   RUNG wire#powerrail
      Contact( #alwaysOn )
      wire#w1
      Contact( #State."Ready For Transfer" )
      Contact( #IN_Dose_Run )
      Contact( #IN_Dose_Valve_Cmd )
      Contact( #IN_Dose_LineOK )
      wire#w2
      Coil( #Actuator.AV_Outlet )
   END_RUNG
   RUNG wire#w1
      Contact( #State."CIP Tank" )
      Contact( #"CIP Request OK" )
   END_RUNG wire#w2
   RUNG wire#w1
      Contact( #Actuator.AV_Outlet )
      Coil( #Out_AV_Outlet )
   END_RUNG
   // the same network as SCL:
   #Actuator.AV_Outlet := #alwaysOn AND ((#State."Ready For Transfer" AND #IN_Dose_Run AND #IN_Dose_Valve_Cmd AND #IN_Dose_LineOK) OR (#State."CIP Tank" AND #"CIP Request OK"));
   #Out_AV_Outlet := #alwaysOn AND #Actuator.AV_Outlet;
END_REGION

REGION Network 17: AV Transfer
   RUNG wire#powerrail
      Contact( #alwaysOn )
      Contact( #Actuator.AV_Transfer )
      Coil( #Out_AV_Transfer )
   END_RUNG
   // the same network as SCL:
   #Out_AV_Transfer := #alwaysOn AND #Actuator.AV_Transfer;
END_REGION

REGION Network 18: AV CIP Tank
   RUNG wire#powerrail
      Contact( #alwaysOn )
      Contact( #State."CIP Tank" )
      Contact( #"CIP Request OK" )
      Coil( #Out_AV_CIP_Tank )
   END_RUNG
   // the same network as SCL:
   #Out_AV_CIP_Tank := #alwaysOn AND #State."CIP Tank" AND #"CIP Request OK";
END_REGION

REGION Network 19: AV CIP Line
   RUNG wire#powerrail
      Contact( #alwaysOn )
      Contact( #State."CIP Line" )
      Contact( #"CIP Request OK" )
      Coil( #Out_AV_CIP_Line )
   END_RUNG
   // the same network as SCL:
   #Out_AV_CIP_Line := #alwaysOn AND #State."CIP Line" AND #"CIP Request OK";
END_REGION

REGION Network 20: Pump Transfer
   RUNG wire#powerrail
      Contact( #alwaysOn )
      wire#w1
      Contact( #State."Ready For Transfer" )
      Move(in := #IN_Dose_Pump_Sp, out1 => #Out_P_Transfer_SP)
   END_RUNG
   RUNG wire#w1
      Contact( #State."CIP Line" )
      Move(in := #Param."CIP Pump SP", out1 => #Out_P_Transfer_SP)
   END_RUNG
   RUNG wire#w1
      Contact( #State."Ready For Transfer" )
      Contact( #IN_Dose_Run )
      Contact( #IN_Dose_Pump_Cmd )
      wire#w2
      Coil( #Actuator.P_Transfer )
   END_RUNG
   RUNG wire#w1
      Contact( #State."CIP Line" )
      Contact( #IN_FBAV_CIP_Line )
      Contact( #"CIP Supply ON" )
      Contact( #"CIP Pulse" )
   END_RUNG wire#w2
   RUNG wire#w1
      Contact( #Actuator.P_Transfer )
      Coil( #Out_P_Transfer )
   END_RUNG
   // the same network as SCL:
   IF #alwaysOn AND #State."Ready For Transfer" THEN #Out_P_Transfer_SP := #IN_Dose_Pump_Sp; END_IF;
   IF #alwaysOn AND #State."CIP Line" THEN #Out_P_Transfer_SP := #Param."CIP Pump SP"; END_IF;
   #Actuator.P_Transfer := #alwaysOn AND ((#State."Ready For Transfer" AND #IN_Dose_Run AND #IN_Dose_Pump_Cmd) OR (#State."CIP Line" AND #IN_FBAV_CIP_Line AND #"CIP Supply ON" AND #"CIP Pulse"));
   #Out_P_Transfer := #alwaysOn AND #Actuator.P_Transfer;
END_REGION

REGION Network 21: Pump CIP Tank
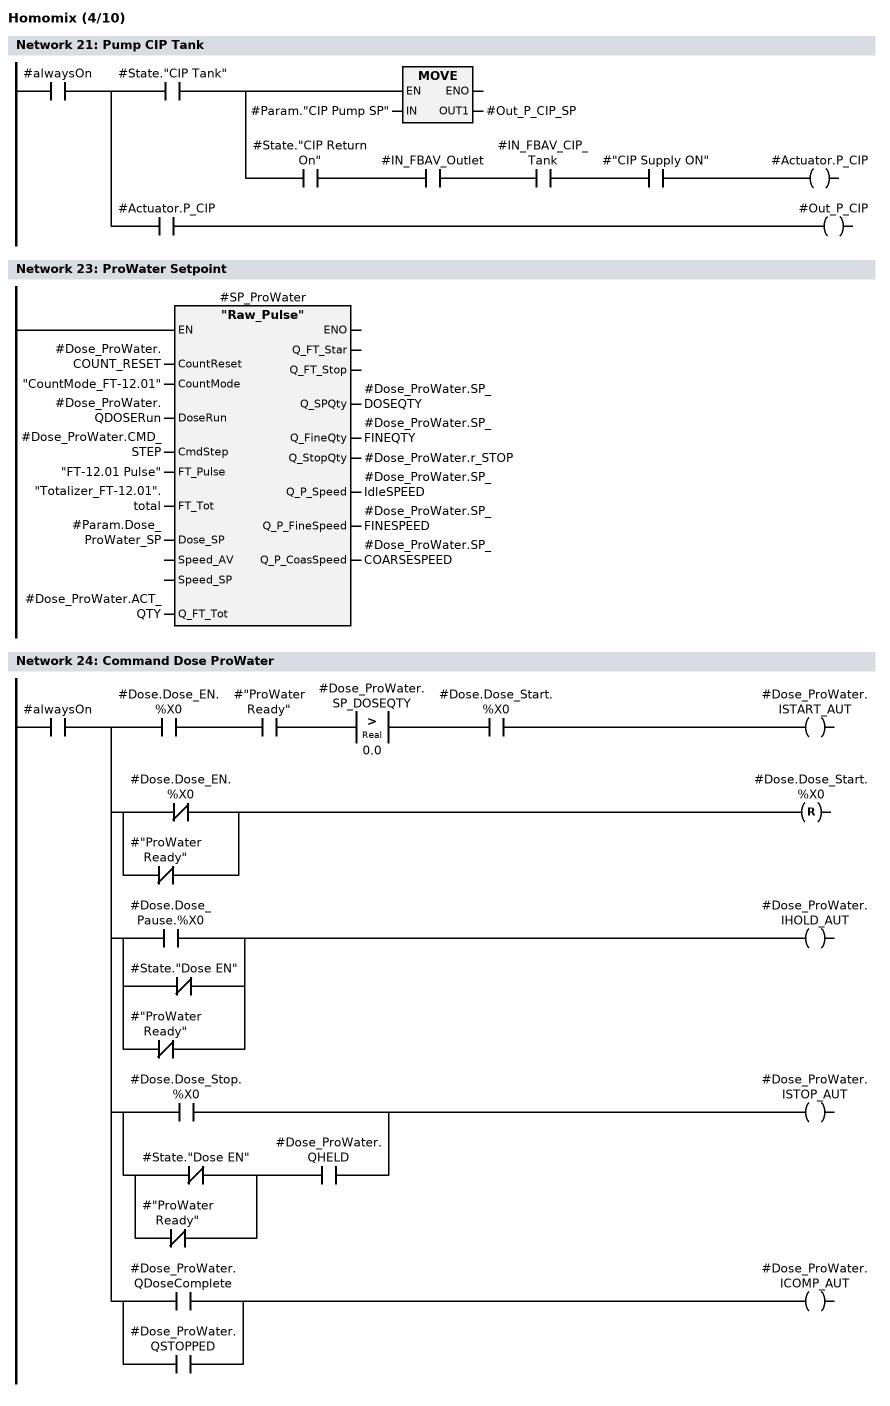
   RUNG wire#powerrail
      Contact( #alwaysOn )
      wire#w1
      Contact( #State."CIP Tank" )
      wire#w2
      Move(in := #Param."CIP Pump SP", out1 => #Out_P_CIP_SP)
   END_RUNG
   RUNG wire#w2
      Contact( #State."CIP Return On" )
      Contact( #IN_FBAV_Outlet )
      Contact( #IN_FBAV_CIP_Tank )
      Contact( #"CIP Supply ON" )
      Coil( #Actuator.P_CIP )
   END_RUNG
   RUNG wire#w1
      Contact( #Actuator.P_CIP )
      Coil( #Out_P_CIP )
   END_RUNG
   // the same network as SCL:
   #_w1 := #alwaysOn AND #State."CIP Tank";
   IF #_w1 THEN #Out_P_CIP_SP := #Param."CIP Pump SP"; END_IF;
   #Actuator.P_CIP := #_w1 AND #State."CIP Return On" AND #IN_FBAV_Outlet AND #IN_FBAV_CIP_Tank AND #"CIP Supply ON";
   #Out_P_CIP := #alwaysOn AND #Actuator.P_CIP;
END_REGION

REGION Network 23: ProWater Setpoint
   RUNG wire#powerrail
      #SP_ProWater(CountReset := #Dose_ProWater.COUNT_RESET, CountMode := "CountMode_FT-12.01", DoseRun := #Dose_ProWater.QDOSERun, CmdStep := #Dose_ProWater.CMD_STEP, FT_Pulse := "FT-12.01 Pulse", FT_Tot := "Totalizer_FT-12.01".total, Dose_SP := #Param.Dose_ProWater_SP, Speed_AV :=, Speed_SP :=, Q_FT_Tot := #Dose_ProWater.ACT_QTY, Q_FT_Star =>, Q_FT_Stop =>, Q_SPQty => #Dose_ProWater.SP_DOSEQTY, Q_FineQty => #Dose_ProWater.SP_FINEQTY, Q_StopQty => #Dose_ProWater.r_STOP, Q_P_Speed => #Dose_ProWater.SP_IdleSPEED, Q_P_FineSpeed => #Dose_ProWater.SP_FINESPEED, Q_P_CoasSpeed => #Dose_ProWater.SP_COARSESPEED)
   END_RUNG
   // the same network as SCL:
   #SP_ProWater(CountReset := #Dose_ProWater.COUNT_RESET,   // "Raw_Pulse"
                CountMode := "CountMode_FT-12.01",
                DoseRun := #Dose_ProWater.QDOSERun,
                CmdStep := #Dose_ProWater.CMD_STEP,
                FT_Pulse := "FT-12.01 Pulse",
                FT_Tot := "Totalizer_FT-12.01".total,
                Dose_SP := #Param.Dose_ProWater_SP,
                Q_FT_Tot := #Dose_ProWater.ACT_QTY,
                Q_SPQty => #Dose_ProWater.SP_DOSEQTY,
                Q_FineQty => #Dose_ProWater.SP_FINEQTY,
                Q_StopQty => #Dose_ProWater.r_STOP,
                Q_P_Speed => #Dose_ProWater.SP_IdleSPEED,
                Q_P_FineSpeed => #Dose_ProWater.SP_FINESPEED,
                Q_P_CoasSpeed => #Dose_ProWater.SP_COARSESPEED);
END_REGION

REGION Network 24: Command Dose ProWater
   RUNG wire#powerrail
      Contact( #alwaysOn )
      wire#w1
      Contact( #Dose.Dose_EN.%X0 )
      Contact( #"ProWater Ready" )
      { S7_Templates := "SrcType := Real" } GT_Contact(in1 := #Dose_ProWater.SP_DOSEQTY, in2 := 0.0)
      Contact( #Dose.Dose_Start.%X0 )
      Coil( #Dose_ProWater.ISTART_AUT )
   END_RUNG
   RUNG wire#w1
      I_Contact( #Dose.Dose_EN.%X0 )
      wire#w2
      R_Coil( #Dose.Dose_Start.%X0 )
   END_RUNG
   RUNG wire#w1
      I_Contact( #"ProWater Ready" )
   END_RUNG wire#w2
   RUNG wire#w1
      Contact( #Dose.Dose_Pause.%X0 )
      wire#w3
      Coil( #Dose_ProWater.IHOLD_AUT )
   END_RUNG
   RUNG wire#w1
      I_Contact( #State."Dose EN" )
   END_RUNG wire#w3
   RUNG wire#w1
      I_Contact( #"ProWater Ready" )
   END_RUNG wire#w3
   RUNG wire#w1
      Contact( #Dose.Dose_Stop.%X0 )
      wire#w4
      Coil( #Dose_ProWater.ISTOP_AUT )
   END_RUNG
   RUNG wire#w1
      I_Contact( #State."Dose EN" )
      wire#w5
      Contact( #Dose_ProWater.QHELD )
   END_RUNG wire#w4
   RUNG wire#w1
      I_Contact( #"ProWater Ready" )
   END_RUNG wire#w5
   RUNG wire#w1
      Contact( #Dose_ProWater.QDoseComplete )
      wire#w6
      Coil( #Dose_ProWater.ICOMP_AUT )
   END_RUNG
   RUNG wire#w1
      Contact( #Dose_ProWater.QSTOPPED )
   END_RUNG wire#w6
   // the same network as SCL:
   #Dose_ProWater.ISTART_AUT := #alwaysOn AND #Dose.Dose_EN.%X0 AND #"ProWater Ready" AND (#Dose_ProWater.SP_DOSEQTY > 0.0) AND #Dose.Dose_Start.%X0;
   IF #alwaysOn AND (NOT #Dose.Dose_EN.%X0 OR NOT #"ProWater Ready") THEN
       #Dose.Dose_Start.%X0 := FALSE;
   END_IF;
   #Dose_ProWater.IHOLD_AUT := #alwaysOn AND (#Dose.Dose_Pause.%X0 OR NOT #State."Dose EN" OR NOT #"ProWater Ready");
   #Dose_ProWater.ISTOP_AUT := #alwaysOn AND (#Dose.Dose_Stop.%X0 OR ((NOT #State."Dose EN" OR NOT #"ProWater Ready") AND #Dose_ProWater.QHELD));
   #Dose_ProWater.ICOMP_AUT := #alwaysOn AND (#Dose_ProWater.QDoseComplete OR #Dose_ProWater.QSTOPPED);
END_REGION

REGION Network 25: Dose ProWater
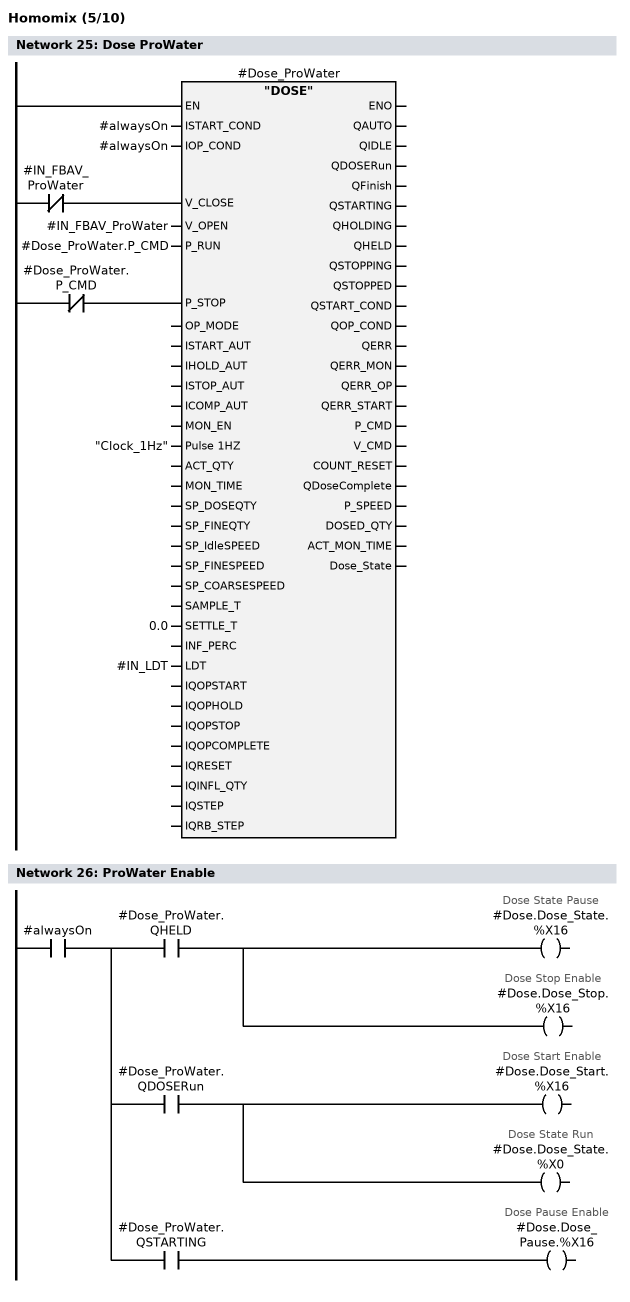
   RUNG wire#powerrail
      #Dose_ProWater(V_CLOSE := wire#w1, P_STOP := wire#w2, ISTART_COND := #alwaysOn, IOP_COND := #alwaysOn, V_OPEN := #IN_FBAV_ProWater, P_RUN := #Dose_ProWater.P_CMD, OP_MODE :=, ISTART_AUT :=, IHOLD_AUT :=, ISTOP_AUT :=, ICOMP_AUT :=, MON_EN :=, "Pulse 1HZ" := "Clock_1Hz", ACT_QTY :=, MON_TIME :=, SP_DOSEQTY :=, SP_FINEQTY :=, SP_IdleSPEED :=, SP_FINESPEED :=, SP_COARSESPEED :=, SAMPLE_T :=, SETTLE_T := 0.0, INF_PERC :=, LDT := #IN_LDT, IQOPSTART :=, IQOPHOLD :=, IQOPSTOP :=, IQOPCOMPLETE :=, IQRESET :=, IQINFL_QTY :=, IQSTEP :=, IQRB_STEP :=, QAUTO =>, QIDLE =>, QDOSERun =>, QFinish =>, QSTARTING =>, QHOLDING =>, QHELD =>, QSTOPPING =>, QSTOPPED =>, QSTART_COND =>, QOP_COND =>, QERR =>, QERR_MON =>, QERR_OP =>, QERR_START =>, P_CMD =>, V_CMD =>, COUNT_RESET =>, QDoseComplete =>, P_SPEED =>, DOSED_QTY =>, ACT_MON_TIME =>, Dose_State =>)
   END_RUNG
   RUNG wire#powerrail
      I_Contact( #IN_FBAV_ProWater )
   END_RUNG wire#w1
   RUNG wire#powerrail
      I_Contact( #Dose_ProWater.P_CMD )
   END_RUNG wire#w2
   // the same network as SCL:
   #Dose_ProWater(ISTART_COND := #alwaysOn,   // "DOSE"
                  IOP_COND := #alwaysOn,
                  V_CLOSE := NOT #IN_FBAV_ProWater,
                  V_OPEN := #IN_FBAV_ProWater,
                  P_RUN := #Dose_ProWater.P_CMD,
                  P_STOP := NOT #Dose_ProWater.P_CMD,
                  "Pulse 1HZ" := "Clock_1Hz",
                  SETTLE_T := 0.0,
                  LDT := #IN_LDT);
END_REGION

REGION Network 26: ProWater Enable
   RUNG wire#powerrail
      Contact( #alwaysOn )
      wire#w1
      Contact( #Dose_ProWater.QHELD )
      wire#w2
      Coil( #Dose.Dose_State.%X16 )   // Dose State Pause
   END_RUNG
   RUNG wire#w2
      Coil( #Dose.Dose_Stop.%X16 )   // Dose Stop Enable
   END_RUNG
   RUNG wire#w1
      Contact( #Dose_ProWater.QDOSERun )
      wire#w3
      Coil( #Dose.Dose_Start.%X16 )   // Dose Start Enable
   END_RUNG
   RUNG wire#w3
      Coil( #Dose.Dose_State.%X0 )   // Dose State Run
   END_RUNG
   RUNG wire#w1
      Contact( #Dose_ProWater.QSTARTING )
      Coil( #Dose.Dose_Pause.%X16 )   // Dose Pause Enable
   END_RUNG
   // the same network as SCL:
   #Dose.Dose_State.%X16 := #alwaysOn AND #Dose_ProWater.QHELD;   // Dose State Pause
   #Dose.Dose_Stop.%X16 := #Dose.Dose_State.%X16;   // Dose Stop Enable
   #Dose.Dose_Start.%X16 := #alwaysOn AND #Dose_ProWater.QDOSERun;   // Dose Start Enable
   #Dose.Dose_State.%X0 := #Dose.Dose_Start.%X16;   // Dose State Run
   #Dose.Dose_Pause.%X16 := #alwaysOn AND #Dose_ProWater.QSTARTING;   // Dose Pause Enable
END_REGION

REGION Network 27: ProWater Header Req and Valve
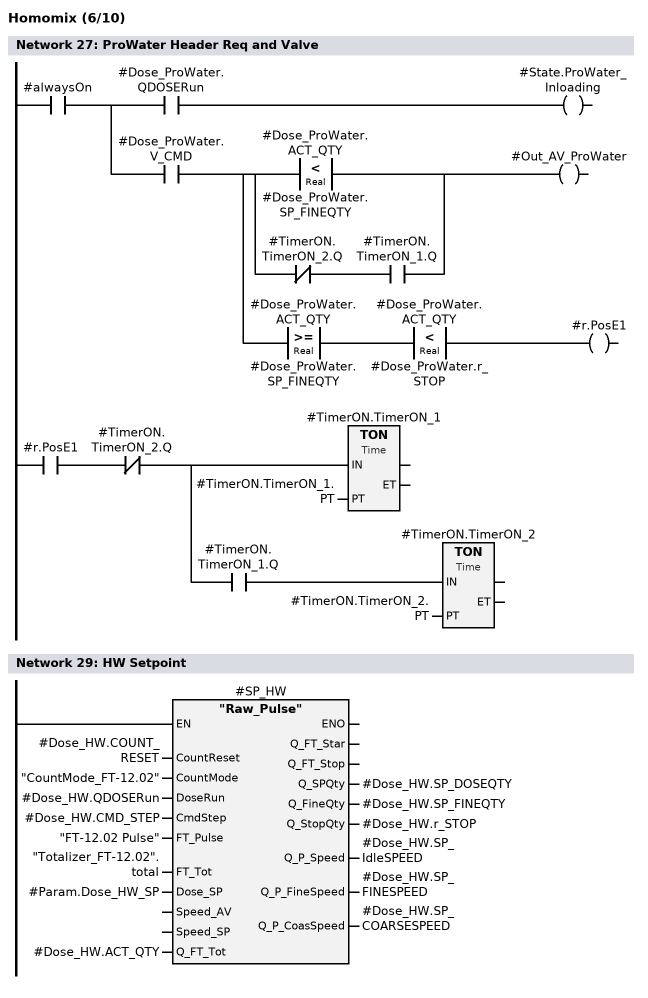
   RUNG wire#powerrail
      Contact( #alwaysOn )
      wire#w1
      Contact( #Dose_ProWater.QDOSERun )
      Coil( #State.ProWater_Inloading )
   END_RUNG
   RUNG wire#w1
      Contact( #Dose_ProWater.V_CMD )
      wire#w2
      { S7_Templates := "SrcType := Real" } LT_Contact(in1 := #Dose_ProWater.ACT_QTY, in2 := #Dose_ProWater.SP_FINEQTY)
      wire#w3
      Coil( #Out_AV_ProWater )
   END_RUNG
   RUNG wire#w2
      I_Contact( #TimerON.TimerON_2.Q )
      Contact( #TimerON.TimerON_1.Q )
   END_RUNG wire#w3
   RUNG wire#w2
      { S7_Templates := "SrcType := Real" } GE_Contact(in1 := #Dose_ProWater.ACT_QTY, in2 := #Dose_ProWater.SP_FINEQTY)
      { S7_Templates := "SrcType := Real" } LT_Contact(in1 := #Dose_ProWater.ACT_QTY, in2 := #Dose_ProWater.r_STOP)
      Coil( #r.PosE1 )
   END_RUNG
   RUNG wire#powerrail
      Contact( #r.PosE1 )
      I_Contact( #TimerON.TimerON_2.Q )
      wire#w4
      { S7_Templates := "time_type := Time" } #TimerON.TimerON_1.TON(pt := #TimerON.TimerON_1.PT, et =>)
   END_RUNG
   RUNG wire#w4
      Contact( #TimerON.TimerON_1.Q )
      { S7_Templates := "time_type := Time" } #TimerON.TimerON_2.TON(pt := #TimerON.TimerON_2.PT, et =>)
   END_RUNG
   // the same network as SCL:
   #State.ProWater_Inloading := #alwaysOn AND #Dose_ProWater.QDOSERun;
   #_w1 := #alwaysOn AND #Dose_ProWater.V_CMD;
   #Out_AV_ProWater := #_w1 AND ((#Dose_ProWater.ACT_QTY < #Dose_ProWater.SP_FINEQTY) OR (NOT #TimerON.TimerON_2.Q AND #TimerON.TimerON_1.Q));
   #r.PosE1 := #_w1 AND (#Dose_ProWater.ACT_QTY >= #Dose_ProWater.SP_FINEQTY) AND (#Dose_ProWater.ACT_QTY < #Dose_ProWater.r_STOP);
   #_w2 := #r.PosE1 AND NOT #TimerON.TimerON_2.Q;
   #TimerON.TimerON_1.TON(IN := #_w2, PT := #TimerON.TimerON_1.PT);
   #TimerON.TimerON_2.TON(IN := #_w2 AND #TimerON.TimerON_1.Q, PT := #TimerON.TimerON_2.PT);
END_REGION

REGION Network 29: HW Setpoint
   RUNG wire#powerrail
      #SP_HW(CountReset := #Dose_HW.COUNT_RESET, CountMode := "CountMode_FT-12.02", DoseRun := #Dose_HW.QDOSERun, CmdStep := #Dose_HW.CMD_STEP, FT_Pulse := "FT-12.02 Pulse", FT_Tot := "Totalizer_FT-12.02".total, Dose_SP := #Param.Dose_HW_SP, Speed_AV :=, Speed_SP :=, Q_FT_Tot := #Dose_HW.ACT_QTY, Q_FT_Star =>, Q_FT_Stop =>, Q_SPQty => #Dose_HW.SP_DOSEQTY, Q_FineQty => #Dose_HW.SP_FINEQTY, Q_StopQty => #Dose_HW.r_STOP, Q_P_Speed => #Dose_HW.SP_IdleSPEED, Q_P_FineSpeed => #Dose_HW.SP_FINESPEED, Q_P_CoasSpeed => #Dose_HW.SP_COARSESPEED)
   END_RUNG
   // the same network as SCL:
   #SP_HW(CountReset := #Dose_HW.COUNT_RESET,   // "Raw_Pulse"
          CountMode := "CountMode_FT-12.02",
          DoseRun := #Dose_HW.QDOSERun,
          CmdStep := #Dose_HW.CMD_STEP,
          FT_Pulse := "FT-12.02 Pulse",
          FT_Tot := "Totalizer_FT-12.02".total,
          Dose_SP := #Param.Dose_HW_SP,
          Q_FT_Tot := #Dose_HW.ACT_QTY,
          Q_SPQty => #Dose_HW.SP_DOSEQTY,
          Q_FineQty => #Dose_HW.SP_FINEQTY,
          Q_StopQty => #Dose_HW.r_STOP,
          Q_P_Speed => #Dose_HW.SP_IdleSPEED,
          Q_P_FineSpeed => #Dose_HW.SP_FINESPEED,
          Q_P_CoasSpeed => #Dose_HW.SP_COARSESPEED);
END_REGION

REGION Network 30: Command Dose HW
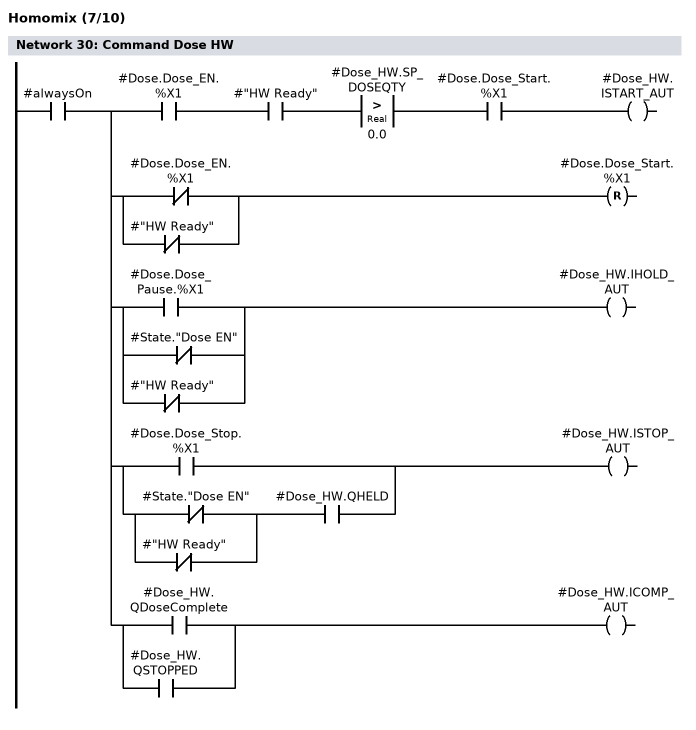
   RUNG wire#powerrail
      Contact( #alwaysOn )
      wire#w1
      Contact( #Dose.Dose_EN.%X1 )
      Contact( #"HW Ready" )
      { S7_Templates := "SrcType := Real" } GT_Contact(in1 := #Dose_HW.SP_DOSEQTY, in2 := 0.0)
      Contact( #Dose.Dose_Start.%X1 )
      Coil( #Dose_HW.ISTART_AUT )
   END_RUNG
   RUNG wire#w1
      I_Contact( #Dose.Dose_EN.%X1 )
      wire#w2
      R_Coil( #Dose.Dose_Start.%X1 )
   END_RUNG
   RUNG wire#w1
      I_Contact( #"HW Ready" )
   END_RUNG wire#w2
   RUNG wire#w1
      Contact( #Dose.Dose_Pause.%X1 )
      wire#w3
      Coil( #Dose_HW.IHOLD_AUT )
   END_RUNG
   RUNG wire#w1
      I_Contact( #State."Dose EN" )
   END_RUNG wire#w3
   RUNG wire#w1
      I_Contact( #"HW Ready" )
   END_RUNG wire#w3
   RUNG wire#w1
      Contact( #Dose.Dose_Stop.%X1 )
      wire#w4
      Coil( #Dose_HW.ISTOP_AUT )
   END_RUNG
   RUNG wire#w1
      I_Contact( #State."Dose EN" )
      wire#w5
      Contact( #Dose_HW.QHELD )
   END_RUNG wire#w4
   RUNG wire#w1
      I_Contact( #"HW Ready" )
   END_RUNG wire#w5
   RUNG wire#w1
      Contact( #Dose_HW.QDoseComplete )
      wire#w6
      Coil( #Dose_HW.ICOMP_AUT )
   END_RUNG
   RUNG wire#w1
      Contact( #Dose_HW.QSTOPPED )
   END_RUNG wire#w6
   // the same network as SCL:
   #Dose_HW.ISTART_AUT := #alwaysOn AND #Dose.Dose_EN.%X1 AND #"HW Ready" AND (#Dose_HW.SP_DOSEQTY > 0.0) AND #Dose.Dose_Start.%X1;
   IF #alwaysOn AND (NOT #Dose.Dose_EN.%X1 OR NOT #"HW Ready") THEN #Dose.Dose_Start.%X1 := FALSE; END_IF;
   #Dose_HW.IHOLD_AUT := #alwaysOn AND (#Dose.Dose_Pause.%X1 OR NOT #State."Dose EN" OR NOT #"HW Ready");
   #Dose_HW.ISTOP_AUT := #alwaysOn AND (#Dose.Dose_Stop.%X1 OR ((NOT #State."Dose EN" OR NOT #"HW Ready") AND #Dose_HW.QHELD));
   #Dose_HW.ICOMP_AUT := #alwaysOn AND (#Dose_HW.QDoseComplete OR #Dose_HW.QSTOPPED);
END_REGION

REGION Network 31: Dose HW
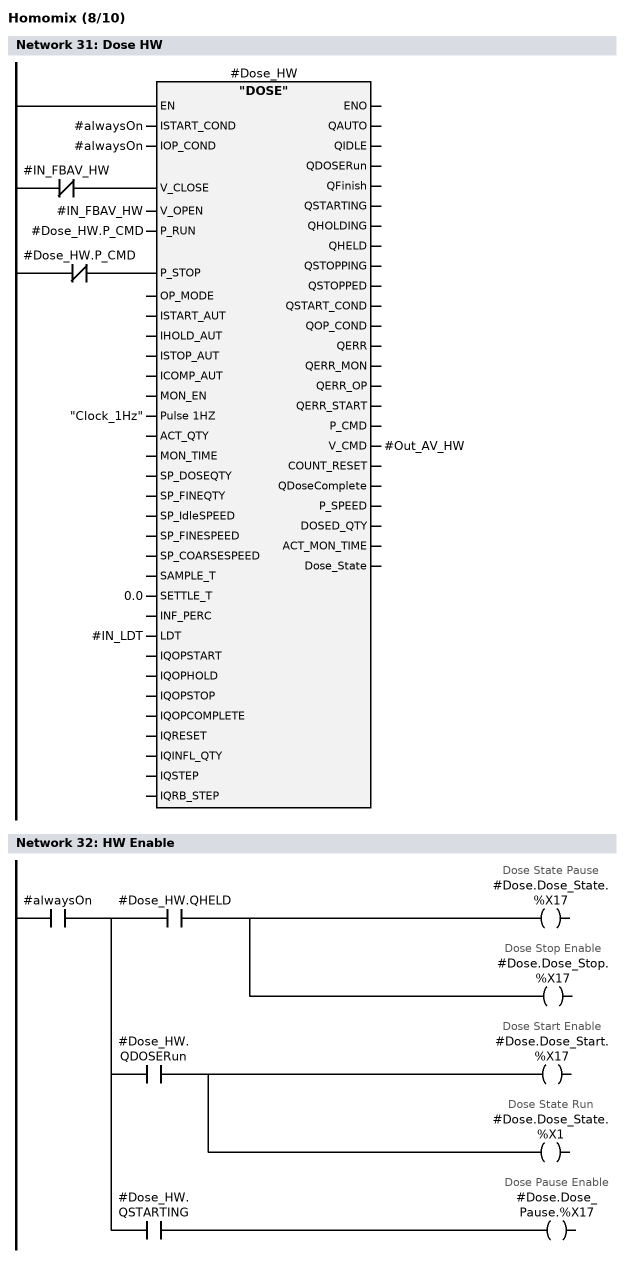
   RUNG wire#powerrail
      #Dose_HW(V_CLOSE := wire#w1, P_STOP := wire#w2, ISTART_COND := #alwaysOn, IOP_COND := #alwaysOn, V_OPEN := #IN_FBAV_HW, P_RUN := #Dose_HW.P_CMD, OP_MODE :=, ISTART_AUT :=, IHOLD_AUT :=, ISTOP_AUT :=, ICOMP_AUT :=, MON_EN :=, "Pulse 1HZ" := "Clock_1Hz", ACT_QTY :=, MON_TIME :=, SP_DOSEQTY :=, SP_FINEQTY :=, SP_IdleSPEED :=, SP_FINESPEED :=, SP_COARSESPEED :=, SAMPLE_T :=, SETTLE_T := 0.0, INF_PERC :=, LDT := #IN_LDT, IQOPSTART :=, IQOPHOLD :=, IQOPSTOP :=, IQOPCOMPLETE :=, IQRESET :=, IQINFL_QTY :=, IQSTEP :=, IQRB_STEP :=, QAUTO =>, QIDLE =>, QDOSERun =>, QFinish =>, QSTARTING =>, QHOLDING =>, QHELD =>, QSTOPPING =>, QSTOPPED =>, QSTART_COND =>, QOP_COND =>, QERR =>, QERR_MON =>, QERR_OP =>, QERR_START =>, P_CMD =>, V_CMD => #Out_AV_HW, COUNT_RESET =>, QDoseComplete =>, P_SPEED =>, DOSED_QTY =>, ACT_MON_TIME =>, Dose_State =>)
   END_RUNG
   RUNG wire#powerrail
      I_Contact( #IN_FBAV_HW )
   END_RUNG wire#w1
   RUNG wire#powerrail
      I_Contact( #Dose_HW.P_CMD )
   END_RUNG wire#w2
   // the same network as SCL:
   #Dose_HW(ISTART_COND := #alwaysOn,   // "DOSE"
            IOP_COND := #alwaysOn,
            V_CLOSE := NOT #IN_FBAV_HW,
            V_OPEN := #IN_FBAV_HW,
            P_RUN := #Dose_HW.P_CMD,
            P_STOP := NOT #Dose_HW.P_CMD,
            "Pulse 1HZ" := "Clock_1Hz",
            SETTLE_T := 0.0,
            LDT := #IN_LDT,
            V_CMD => #Out_AV_HW);
END_REGION

REGION Network 32: HW Enable
   RUNG wire#powerrail
      Contact( #alwaysOn )
      wire#w1
      Contact( #Dose_HW.QHELD )
      wire#w2
      Coil( #Dose.Dose_State.%X17 )   // Dose State Pause
   END_RUNG
   RUNG wire#w2
      Coil( #Dose.Dose_Stop.%X17 )   // Dose Stop Enable
   END_RUNG
   RUNG wire#w1
      Contact( #Dose_HW.QDOSERun )
      wire#w3
      Coil( #Dose.Dose_Start.%X17 )   // Dose Start Enable
   END_RUNG
   RUNG wire#w3
      Coil( #Dose.Dose_State.%X1 )   // Dose State Run
   END_RUNG
   RUNG wire#w1
      Contact( #Dose_HW.QSTARTING )
      Coil( #Dose.Dose_Pause.%X17 )   // Dose Pause Enable
   END_RUNG
   // the same network as SCL:
   #Dose.Dose_State.%X17 := #alwaysOn AND #Dose_HW.QHELD;   // Dose State Pause
   #Dose.Dose_Stop.%X17 := #Dose.Dose_State.%X17;   // Dose Stop Enable
   #Dose.Dose_Start.%X17 := #alwaysOn AND #Dose_HW.QDOSERun;   // Dose Start Enable
   #Dose.Dose_State.%X1 := #Dose.Dose_Start.%X17;   // Dose State Run
   #Dose.Dose_Pause.%X17 := #alwaysOn AND #Dose_HW.QSTARTING;   // Dose Pause Enable
END_REGION

REGION Network 33: HW Header Req and Valve
